END_FUNCTION_BLOCK

FUNCTION "FC_TPConveyorMapping" : Void
{ S7_Optimized_Access := 'TRUE' }
VERSION : 0.1
// ATTRIBUTES
// AUTO_NUMBER = True
// BLOCK_NUMBER = 30
// END_ATTRIBUTES
   VAR_INPUT
      iUDT_ConveyorStatus : "UDT_ConveyorStatus";
      iv_VfdStatus : Variant;
      iUDT_ConveyorInterface : "UDT_ConveyorInterface";
      iUDT_ConveyorConfiguration : "UDT_ConveyorConfiguration";
      is_ConveyorID : String;
   END_VAR

   VAR_OUTPUT
      qUDT_TPConveyorStatus : "UDT_ConveyorStatus";
      qUDT_TPConveyorInterface : "UDT_ConveyorInterface";
      qUDT_TPCommandState : "UDT_ConveyorCommand";   // Actual state of conveyor commands in DB_HMICommands
      qUDT_TPConveyorConfiguration : "UDT_ConveyorConfiguration";
      qs_TPSelectedConveyorName : String;
   END_VAR

   VAR_IN_OUT
      iqUDT_TPCommandButton : "UDT_TPManualControlButtons";
      iqUDT_ConveyorCommand : "UDT_ConveyorCommand";
      qUDT_TPVfdStatus : "UDT_VfdStatus";
   END_VAR

   VAR_TEMP
      tUDT_VfdStatus : "UDT_VfdStatus";
      tUDT_Ai2Status : "UDT_AixPlcFull4McoStatus";
      temp_ret_val : Int;
   END_VAR


BEGIN
	(*
	----------------------------------------------------------------------------------------

	Version history:
	Date        | Version   | Author        | Remark
	----------------------------------------------------------------------------------------
	18/10/2021  | 1.0       | S.Theocharis  | first release MHS TIA 16
	20/10/2021  | 1.1       | S.Theocharis  | change udt vfd status to variant
	03/06/2022  | 1.2       | M.Krystek     | change MOVE_BLK_VARIANT parameters
	21/02/2023  | 4.0       | F.Baten       | 4.0 Release TIA 17.5
	*)

	REGION 1 - Command Start

	    IF #iqUDT_TPCommandButton.ManualStart THEN
	        #iqUDT_ConveyorCommand.ManualStartStop := TRUE;
	        #iqUDT_TPCommandButton.ManualStart := False;
	    END_IF;

	END_REGION

	REGION 2 - Command Stop

	    IF #iqUDT_TPCommandButton.ManualStop THEN
	        #iqUDT_ConveyorCommand.ManualStartStop := FALSE;
	        #iqUDT_TPCommandButton.ManualStop := False;
	    END_IF;
	END_REGION

	REGION 3 - Command Nominal Speed

	    IF #iqUDT_TPCommandButton.ManualFullSpeed THEN
	        #iqUDT_ConveyorCommand.ManualFullSpeed := TRUE;
	        #iqUDT_TPCommandButton.ManualFullSpeed := False;
	    END_IF;
	END_REGION

	REGION 4 - Command Low Speed

	    IF #iqUDT_TPCommandButton.ManualLowSpeed THEN
	        #iqUDT_ConveyorCommand.ManualFullSpeed := FALSE;
	        #iqUDT_TPCommandButton.ManualLowSpeed := False;
	    END_IF;
	END_REGION

	REGION 5 - Command Reverse

	    IF #iqUDT_TPCommandButton.ManualReverse THEN
	        #iqUDT_ConveyorCommand.Reverse := NOT #iqUDT_ConveyorCommand.Reverse;
	        #iqUDT_ConveyorCommand.ManualStartStop := FALSE; //Stop always to avoid on the fly reverse
	        #iqUDT_TPCommandButton.ManualReverse := False;
	    END_IF;
	END_REGION

	REGION 6 - Command jog

	    #iqUDT_ConveyorCommand.ManualJog := #iqUDT_TPCommandButton.ManualJog;

	    IF #iqUDT_TPCommandButton.ManualJog THEN
	        #iqUDT_ConveyorCommand.ManualStartStop := FALSE;
	    END_IF;

	END_REGION

	REGION 7 - Status

	    #qUDT_TPCommandState := #iqUDT_ConveyorCommand;  //actual status of conveyor commands

	    #qUDT_TPConveyorStatus := #iUDT_ConveyorStatus; //conveyor status

	    //VFD status. Ignore Pulse roller
	    IF TypeOf(#iv_VfdStatus) = TypeOf(#tUDT_VfdStatus) THEN

	        #temp_ret_val := MOVE_BLK_VARIANT(SRC := #iv_VfdStatus,
	                                          COUNT := 1,
	                                          SRC_INDEX := 0,
	                                          DEST_INDEX := 0,
	                                          DEST => #qUDT_TPVfdStatus);

	    ELSE
	        #tUDT_VfdStatus.ErrorCode := #tUDT_VfdStatus.SubErrorCode := 0;
	        #qUDT_TPVfdStatus := #tUDT_VfdStatus;

	    END_IF;

	    //#q_TP_VFDStatus := #i_VFDStatus;

	    #qUDT_TPConveyorInterface := #iUDT_ConveyorInterface; //conveyor interface

	    #qs_TPSelectedConveyorName := #is_ConveyorID; //conveyor ID

	    #qUDT_TPConveyorConfiguration.Bi_Directional_Enable := #iUDT_ConveyorConfiguration.Bi_Directional_Enable; //read only bi directional enable bit from configuration


	END_REGION

END_FUNCTION

FUNCTION_BLOCK "FB_Induct"
TITLE = FB_Induct
{ S7_Optimized_Access := 'TRUE' }
AUTHOR : MHSE
FAMILY : Equipment
VERSION : 3.0
// ATTRIBUTES
// AUTO_NUMBER = True
// BLOCK_NUMBER = 14
// END_ATTRIBUTES
//Function block to control inducting the parcels to a merge conveyor
   VAR_INPUT
      iUDT_InductConfig { ExternalAccessible := 'False'; ExternalVisible := 'False'; ExternalWritable := 'False'} : "UDT_InductConfiguration";   //       Induct configuration parameters
      iUDT_MergeGenConfig { ExternalAccessible := 'False'; ExternalVisible := 'False'; ExternalWritable := 'False'} : "UDT_MergeGeneratorConfig";   //       Merge generator configuration parameters
      iUDT_MergeConvConfig { ExternalAccessible := 'False'; ExternalVisible := 'False'; ExternalWritable := 'False'} : "UDT_ConveyorCommonConfiguration";   //       Merge conveyor common configuration parameters
      iUDT_InductConvConfig { ExternalAccessible := 'False'; ExternalVisible := 'False'; ExternalWritable := 'False'} : "UDT_ConveyorConfiguration";   //       Induct conveyor configuration parameters
      iUDT_InductConvCommonStatus { ExternalAccessible := 'False'; ExternalVisible := 'False'; ExternalWritable := 'False'} : "UDT_CommonStatus";
      idi_PECEoSDistance { ExternalAccessible := 'False'; ExternalVisible := 'False'; ExternalWritable := 'False'} : DInt;   //       Distance between photo eye and the end of conveyor [mm]
      ii_Gin { ExternalAccessible := 'False'; ExternalVisible := 'False'; ExternalWritable := 'False'} : Int;   //       GIN from induct at photoeye position
      ix_SafetyOk { ExternalAccessible := 'False'; ExternalVisible := 'False'; ExternalWritable := 'False'} : Bool;   //       Safety is ok
      ix_inductEnable { ExternalAccessible := 'False'; ExternalVisible := 'False'; ExternalWritable := 'False'} : Bool := TRUE;   //      Enable the induct to make request
      ix_TrackingClear { ExternalAccessible := 'False'; ExternalVisible := 'False'; ExternalWritable := 'False'} : Bool;   //   Tracking area is clear of parcels
   END_VAR

   VAR_OUTPUT
      qx_ExternalRequestDieBack { ExternalAccessible := 'False'; ExternalVisible := 'False'; ExternalWritable := 'False'} : Bool;   // External request dieback
      qx_EnableAutoRecovey { ExternalAccessible := 'False'; ExternalVisible := 'False'; ExternalWritable := 'False'} : Bool;   // Request to enable auto recovery
   END_VAR

   VAR_IN_OUT
      iqs_TrackingData : Array[*] of Int;   //       Tracking data
      iqUDT_Merge : "UDT_Merge";   //       Gapgeneration data
      iqUDT_MergeInterface : "UDT_ConveyorInterface";
      iqUDT_InductInterface : "UDT_ConveyorInterface";
      iqUDT_HandShake : "UDT_ConveyorHandshake";
      iqa_ActualTimeData : Struct
         Offset : Int;
         Max_number_of_records : Int;
         Data {InstructionName := 'DTL'; LibVersion := '1.0'} : Array[0..99] of DTL;
      END_STRUCT;
   END_VAR

   VAR
      sR_TRIG_Displacement {InstructionName := 'R_TRIG'; LibVersion := '1.0'; ExternalAccessible := 'False'; ExternalVisible := 'False'; ExternalWritable := 'False'; S7_SetPoint := 'False'} : R_TRIG;   //       Signal rising edge displacement changed
      sR_TRIG_SetDelay {InstructionName := 'R_TRIG'; LibVersion := '1.0'; ExternalAccessible := 'False'; ExternalVisible := 'False'; ExternalWritable := 'False'; S7_SetPoint := 'False'} : R_TRIG;   //       Signal rising edge of parcel entering
      sR_TRIG_TIP {InstructionName := 'R_TRIG'; LibVersion := '1.0'; ExternalAccessible := 'False'; ExternalVisible := 'False'; ExternalWritable := 'False'; S7_SetPoint := 'False'} : R_TRIG;
      sR_TRIG_Enable {InstructionName := 'R_TRIG'; LibVersion := '1.0'; ExternalAccessible := 'False'; ExternalVisible := 'False'; ExternalWritable := 'False'; S7_SetPoint := 'False'} : R_TRIG;   //   Rising Edge of  Induct Enable signal
      sF_TRIG_sx_Parcel {InstructionName := 'F_TRIG'; LibVersion := '1.0'; ExternalAccessible := 'False'; ExternalVisible := 'False'; ExternalWritable := 'False'; S7_SetPoint := 'False'} : F_TRIG;   // Falling Trigger of sx_Parcel
      sdi_DelayReactivateReq { ExternalAccessible := 'False'; ExternalVisible := 'False'; ExternalWritable := 'False'} : DInt;   //       Actual counter delaying the reactivation request
      sdi_RunningEmpty { ExternalAccessible := 'False'; ExternalVisible := 'False'; ExternalWritable := 'False'} : DInt;   //       Actual counter distance running empty
      si_RequestLength { ExternalAccessible := 'False'; ExternalVisible := 'False'; ExternalWritable := 'False'} : Int;   //       Calculated length to be requested
      si_GINlength { ExternalAccessible := 'False'; ExternalVisible := 'False'; ExternalWritable := 'False'} : Int;   //       Length found in GIN DN or set beacuse of invalid length
      si_Gaplength { ExternalAccessible := 'False'; ExternalVisible := 'False'; ExternalWritable := 'False'} : Int;   //       Length for this parcel
      si_ArrayLengthFlexGap { ExternalAccessible := 'False'; ExternalVisible := 'False'; ExternalWritable := 'False'} : Int;   //       Size of the flexGapsize
      si_ArrayLengthTracking { ExternalAccessible := 'False'; ExternalVisible := 'False'; ExternalWritable := 'False'} : Int;   //       Size of the tracking array
      si_ArrayLengthFIFO { ExternalAccessible := 'False'; ExternalVisible := 'False'; ExternalWritable := 'False'} : Int;   //       Size of the FIFO
      si_DistanceToEnd { ExternalAccessible := 'False'; ExternalVisible := 'False'; ExternalWritable := 'False'} : Int;   //       Parcels distance to end of induct conveyor
      si_InductPoint { ExternalAccessible := 'False'; ExternalVisible := 'False'; ExternalWritable := 'False'} : Int;   //       Calculated induct point
      si_StartSearch { ExternalAccessible := 'False'; ExternalVisible := 'False'; ExternalWritable := 'False'} : Int;   //       Value declaring the start of the search area
      si_EndSearch { ExternalAccessible := 'False'; ExternalVisible := 'False'; ExternalWritable := 'False'} : Int;   //       Value declaring the end of the search area
      si_LoopCountFlexgap { ExternalAccessible := 'False'; ExternalVisible := 'False'; ExternalWritable := 'False'} : Int;   //       Loopcounter searching in configuration for a match for the parcellength
      si_LoopCountGapSearch { ExternalAccessible := 'False'; ExternalVisible := 'False'; ExternalWritable := 'False'} : Int;   //       Loopcounter searching in Trackingdata for a gap
      si_LoopCountCodeSearch { ExternalAccessible := 'False'; ExternalVisible := 'False'; ExternalWritable := 'False'} : Int;   //       Loopcounter searching for code -100
      si_LoopCountSyncSearch { ExternalAccessible := 'False'; ExternalVisible := 'False'; ExternalWritable := 'False'} : Int;   //       Loopcounter searching for code -100
      si_LoopCountFIFOSearch { ExternalAccessible := 'False'; ExternalVisible := 'False'; ExternalWritable := 'False'} : Int;   //       Loopcounter searching FIFO for request to remove
      si_LoopCountWriteGIN { ExternalAccessible := 'False'; ExternalVisible := 'False'; ExternalWritable := 'False'} : Int;   //       Loopcounter to write the GIN for the length of the parcel
      si_LastGIN { ExternalAccessible := 'False'; ExternalVisible := 'False'; ExternalWritable := 'False'} : Int;   //       Last processed GIN
      si_Flexgap { ExternalAccessible := 'False'; ExternalVisible := 'False'; ExternalWritable := 'False'} : Int;   //       Found flexible gapsize [cm]
      si_PosDataInSearchArea { ExternalAccessible := 'False'; ExternalVisible := 'False'; ExternalWritable := 'False'} : Int;   //       Length to wait to search for a gap
      si_WritePosition { ExternalAccessible := 'False'; ExternalVisible := 'False'; ExternalWritable := 'False'} : Int;   //       Position to write to in tracking
      si_Syncdifference { ExternalAccessible := 'False'; ExternalVisible := 'False'; ExternalWritable := 'False'} : Int;   //       Difference in positions pec and tracking
      si_SyncDistance { ExternalAccessible := 'False'; ExternalVisible := 'False'; ExternalWritable := 'False'} : Int;   //       Distance to perform the synchronisation in
      si_MergeRunLength { ExternalAccessible := 'False'; ExternalVisible := 'False'; ExternalWritable := 'False'} : Int;   //     Distance the merge conveyor has run when Inudct is waiting
      si_DelayDiebackLength { ExternalAccessible := 'False'; ExternalVisible := 'False'; ExternalWritable := 'False'} : Int;   //     length Run before applying die back [cm]
      si_TrackingPointer { ExternalAccessible := 'False'; ExternalVisible := 'False'; ExternalWritable := 'False'} : Int;   //   Tracking poitner to search in the tracking
      sx_Sync { ExternalAccessible := 'False'; ExternalVisible := 'False'; ExternalWritable := 'False'} : Bool;   //       Code search to synchronise
      sx_ConfigError { ExternalAccessible := 'False'; ExternalVisible := 'False'; ExternalWritable := 'False'} : Bool;   //       Error in the configuration
      sx_FindLength { ExternalAccessible := 'False'; ExternalVisible := 'False'; ExternalWritable := 'False'} : Bool;   //       Find the length of the new parcel
      sx_Parcel { ExternalAccessible := 'False'; ExternalVisible := 'False'; ExternalWritable := 'False'} : Bool;   //       The parcel is present an not yet handled completely
      sx_GapRequested { ExternalAccessible := 'False'; ExternalVisible := 'False'; ExternalWritable := 'False'} : Bool;   //       The request is done for the latest parcel
      sx_SearchGapInTracking { ExternalAccessible := 'False'; ExternalVisible := 'False'; ExternalWritable := 'False'} : Bool;   //       True = Search for space in tracking to induct without merge generation
      sx_LastCodeNeg { ExternalAccessible := 'False'; ExternalVisible := 'False'; ExternalWritable := 'False'} : Bool;   //       True = Last found code was a negative one
      sx_FreeGapAvailable { ExternalAccessible := 'False'; ExternalVisible := 'False'; ExternalWritable := 'False'} : Bool;   //       There is a free space found, big enough to insert the parcel
      sx_ValidWindowCodeFound { ExternalAccessible := 'False'; ExternalVisible := 'False'; ExternalWritable := 'False'} : Bool;   //       There is a valid window code found
      sx_CodeAtposition { ExternalAccessible := 'False'; ExternalVisible := 'False'; ExternalWritable := 'False'} : Bool;
      sx_InductEnable { ExternalAccessible := 'False'; ExternalVisible := 'False'; ExternalWritable := 'False'} : Bool;   //       The parcel is enabled to induct
      sx_DiebackInductConveyor { ExternalAccessible := 'False'; ExternalVisible := 'False'; ExternalWritable := 'False'} : Bool;   //       Memory to stop the induct conveyor
      sx_Hold { ExternalAccessible := 'False'; ExternalVisible := 'False'; ExternalWritable := 'False'} : Bool;   //       Hold inducting
      sx_Active { ExternalAccessible := 'False'; ExternalVisible := 'False'; ExternalWritable := 'False'} : Bool;
      sx_EnableAutoRecovery { ExternalAccessible := 'False'; ExternalVisible := 'False'; ExternalWritable := 'False'} : Bool;   //     Enable Auto Recovery for Induct
      sx_RecoveryRequest { ExternalAccessible := 'False'; ExternalVisible := 'False'; ExternalWritable := 'False'} : Bool;
   END_VAR

   VAR CONSTANT
      ci_SearchArea : Int := 3;
   END_VAR


BEGIN
	(*
	----------------------------------------------------------------------------------------

	Version history:
	Date        | Version   | Author        | Remark
	----------------------------------------------------------------------------------------
	24/09/2019  | 1.0       | F.Baten       | first release TIA 15.1
	31/10/2019  | 1.1       | F.Baten       | qi_SpeedSetpoint changed to int because of conveyor interface change
	12/11/2019  | 3.0       | P.Majka       | 3.0 MHS library release TIA 15.1
	07/01/2020  | 3.1       | F.Baten       | Changed RequestInFifo to be handshaking
	                                        | Merged region 4.3 and 4.4
	09/01/2020  | 3.2       | F.Baten       | Removed speed calculation
	14/01/2020  | 3.3       | F.Baten       | Removed global FIFO full signal as it was not generated and made it local
	14/01/2020  | 3.4       | F.Baten       | Changed displacement detection equal to 0 and not to be 1 as it can also be bigger
	            | 3.5       |               | Renamed ii_PEC_EoSDistance to idi_PEC_EoSDistance
	15/01/2020  | 3.6       | L.Klar        | GIN record structure updated, parcel length remapped
	23/01/2020  | 3.7       | F.Baten       | Added reset when parcel is at end of conveyor but for some reason not detected
	                                          Modified dieback: alsways goto dieback when parcel is handled
	18/02/2020  | 3.8       | F.Baten       | Modified "Search 1: Gap '0'" , added +1 to wait to search again.
	15/10/2020  | 3.9       | F.Baten       | Reqactivation request: added if active to keep active
	                                          removed displacement check out of search
	20/05/2021  | 3.10      | M.Singh       | Enabled Auto Recovery based on the displacemt on Merge
	20/04/2022  | 3.11      | M.Piela       | Added Auto recovery output
	24/05/2022  | 3.12      | M.Roijen      | Changed FOR loop region 5.2 copy gin to tracking (add -1).
	22/07/2022  | 3.13      | M.Piela       | Reset the sx_Active and set dieback induct on falling edge of sx_Parcel instead of rising edge of TIP.
	21/02/2023  | 4.0       | F.Baten       | 4.0 Release TIA 17.5
	*)

	REGION 1 - New GIN received
	    // When the new GIN is received:
	    // - first save the GIN and set/reset statuses
	    // - calculate the requested length for this parcel
	    // - requeset a gap for this parcel

	    REGION 1.1 - New gin received is NOT equal TO '0' AND NOT equal TO last gin
	        //#s_R_TRIG_TIP(CLK := #iq_UDT_HandShake.TIP);
	        // IF #ii_Gin <> 0 AND #ii_Gin <> #si_LastGIN AND NOT #iq_UDT_HandShake.TIP AND NOT #s_F_TRIG_TIP.Q

	        IF #ii_Gin <> 0 AND #ii_Gin <> #si_LastGIN AND #ix_inductEnable
	        THEN
	            #sx_FindLength := FALSE;                                                    // To set length for a flexible gap
	            #sx_GapRequested := FALSE;                                                  // To initiate length calculation for gap and request the gap to FIFO
	            #sx_DiebackInductConveyor := TRUE;                                             // Activate dieback to stop the conveyor while waiting on a gap
	            #sx_Sync := FALSE;                                                          // Sync speed is not calculated
	            #sx_Parcel := TRUE;                                                         // Activate the induct search
	            #sx_Active := TRUE;                                                         // The parcel is not transferred to the next conveyor
	            #si_LastGIN := #ii_Gin;                                                     // Memorise
	            #si_DistanceToEnd := DINT_TO_INT(#idi_PECEoSDistance) / 10;                // Actual distance to end (in tracking array units)
	            #si_GINlength := DINT_TO_INT("DB_GIN".GIN[#si_LastGIN].General.Length);     // set length
	            IF #si_GINlength = 0
	            THEN
	                #si_GINlength := #iUDT_InductConfig.MaxParcelSize / 10;
	            END_IF;

	            IF #sx_RecoveryRequest
	            THEN

	                #si_DistanceToEnd := #iUDT_InductConfig.ParcelStopPositionAutoRecovery;                                                     // Actual distance to end (in tracking array units)
	                #si_GINlength := (#iUDT_InductConfig.MaxParcelSize / 10) + #iUDT_InductConfig.RecoveryAdditionalGap;
	                #sx_RecoveryRequest := FALSE;
	            END_IF;

	        END_IF;

	        // There is a parcel on the inductconveyor but it had no GIN (not even UFO)
	        IF (#iqUDT_HandShake.RTS                                                       // If Induct is ready to Send
	            OR #iUDT_InductConvCommonStatus.Dieback)                                   // Or is in die back
	            AND NOT #sx_Active                                                          // And Induct is not active
	            AND #ix_inductEnable
	        THEN
	            #si_MergeRunLength := #si_MergeRunLength - #iqUDT_MergeInterface.Displacement;
	        ELSE
	            #si_MergeRunLength := #iUDT_InductConfig.DistanceRunBeforeAutoRecovery;
	        END_IF;

	        #sx_EnableAutoRecovery := FALSE;

	        IF #si_MergeRunLength <= 0
	        THEN
	            #sx_EnableAutoRecovery := True;
	            #si_MergeRunLength := #iUDT_InductConfig.DistanceRunBeforeAutoRecovery;
	        END_IF;

	        #sR_TRIG_Enable(CLK := #ix_inductEnable);

	        IF #sx_EnableAutoRecovery                                                     // Make a new request to autorecover
	            OR (#sR_TRIG_Enable.Q
	            AND NOT #ix_TrackingClear)
	        THEN
	            #sx_FindLength := FALSE;                                                    // To set length for a flexible gap
	            #sx_GapRequested := FALSE;                                                  // To initiate length calculation for gap and request the gap to FIFO
	            #sx_DiebackInductConveyor := TRUE;                                             // Activate dieback to stop the conveyor while waiting on a gap
	            #sx_Sync := FALSE;                                                          // Sync speed is not calculated
	            #sx_Parcel := TRUE;                                                         // Activate the induct search
	            #sx_Active := TRUE;                                                         // The parcel is not transferred to the next conveyor
	            #si_LastGIN := -50;                                                         // Memorise
	            #si_DistanceToEnd := #iUDT_InductConfig.ParcelStopPositionAutoRecovery;                                                     // Actual distance to end (in tracking array units)
	            #si_GINlength := (#iUDT_InductConfig.MaxParcelSize / 10) + #iUDT_InductConfig.RecoveryAdditionalGap;
	            #sx_RecoveryRequest := TRUE;



	            // temp code
	            #iqa_ActualTimeData.Data[#iqa_ActualTimeData.Offset] := "DB_Time".ActualTimeDTL;
	            #iqa_ActualTimeData.Offset := #iqa_ActualTimeData.Offset + 1;
	        END_IF;

	        #qx_EnableAutoRecovey := #sx_EnableAutoRecovery;

	        IF #iqa_ActualTimeData.Offset = #iqa_ActualTimeData.Max_number_of_records
	        THEN
	            #iqa_ActualTimeData.Offset := 1;
	        END_IF;


	    END_REGION

	    REGION 1.2 - Calculate the required gap depending on the mode
	        CASE #iUDT_InductConfig.GapMode OF

	            1:  // Gap is Head to head
	                #si_RequestLength := #iUDT_InductConfig.GapHeadToHead;
	                #si_Gaplength := #si_RequestLength - #si_GINlength;
	                #sx_FindLength := TRUE;                                                 // New GIN length is set

	            2:  // Gap is parcel length + tail to head (fixed)
	                #si_RequestLength := #si_GINlength + #iUDT_InductConfig.GapTailToHead;
	                #si_Gaplength := #iUDT_InductConfig.GapTailToHead;
	                #sx_FindLength := TRUE;                                                 // New GIN length is set

	            3:  // Gap is parcel length + gap depending on length of parcel
	                IF NOT #sx_FindLength
	                THEN
	                    #si_ArrayLengthFlexGap := "FC_GetNrOfArrayEl"(#iUDT_InductConfig.FlexGap); // Determine size of search area
	                    FOR #si_LoopCountFlexgap := 1 TO #si_ArrayLengthFlexGap BY 1 DO                   // Set the loopcounter
	                        #si_Flexgap := #iUDT_InductConfig.MinParcelSize / 10;      // set minimal gapsize
	                        IF #si_GINlength < #iUDT_InductConfig.FlexGap[#si_LoopCountFlexgap]."Maximal length"
	                        THEN
	                            #si_Flexgap := #iUDT_InductConfig.FlexGap[#si_LoopCountFlexgap].Gap;
	                            EXIT;
	                        END_IF;
	                    END_FOR;
	                    #sx_FindLength := TRUE;                                             // New GIN length is calculated
	                END_IF;
	                #si_RequestLength := #si_GINlength + #si_Flexgap;
	                #si_Gaplength := #si_Flexgap;
	                ;

	        END_CASE;
	    END_REGION

	    REGION 1.3 - General
	        // When the transfer is finished set the induct to dieback

	        // IF #s_R_TRIG_TIP.Q  AND NOT #sx_Parcel
	        IF #sF_TRIG_sx_Parcel.Q
	        THEN
	            //     #si_DelayDiebackLength := #i_UDT_InductConfig.MinParcelSize;

	            // END_IF;

	            // IF #si_DelayDiebackLength > 0
	            // THEN
	            //     #si_DelayDiebackLength := #si_DelayDiebackLength - #iq_UDT_InductInterface.Displacement;
	            // END_IF;
	            // IF #si_DelayDiebackLength <= 0
	            // THEN
	            #sx_DiebackInductConveyor := TRUE;                                             // Activate dieback to stop the conveyor while waiting on a gap
	            #sx_Active := FALSE;                                                            // The parcel is now transferred to the next conveyor
	        END_IF;
	        //  #s_R_TRIG_TIP(CLK := #iq_UDT_HandShake.TIP);
	        #sF_TRIG_sx_Parcel(CLK := #sx_Parcel);
	        // When safety is not ok, load the run empty distance
	        IF NOT #ix_SafetyOk
	        THEN
	            #sdi_RunningEmpty := #iUDT_InductConfig.RunEmptyDistance;
	        END_IF;

	        // Hold inducting functions while mergeconveyor runs empty
	        #sx_Hold := (#sdi_RunningEmpty <> 0);

	        // Check every change of the merge conveyor's displacement
	        #sR_TRIG_Displacement(CLK := #iqUDT_MergeInterface.Displacement = 0);             // The merge conveyor has had displacement
	    END_REGION
	END_REGION

	REGION 2 - Request
	    REGION 2.1 - FIFO request
	        // request gap/window for induct
	        IF #sx_Parcel
	            AND NOT #sx_Hold                                                            // Holding all actions
	            AND NOT #sx_GapRequested                                                    // Gap is NOT requested
	            AND NOT #iqUDT_Merge.RequestInFIFO[#iUDT_InductConfig.Induct_Number]      // Requeset is in FIFO
	            AND NOT #iqUDT_Merge.GenerationInactive                                    // Generation is active
	            AND NOT #iUDT_InductConfig.SearchOnly                                      // Only searching for a gap
	            AND NOT (#iqUDT_Merge.LastUsed = #iqUDT_Merge.MaxNumberofEntries)         // The FIFO is full
	        THEN
	            #iqUDT_Merge.LastUsed += 1;                                                // Increase
	            #iqUDT_Merge.RequestInFIFO[#iUDT_InductConfig.Induct_Number] := TRUE;     // Memorise
	            #iqUDT_Merge.FIFO[#iqUDT_Merge.LastUsed].InductNumber := #iUDT_InductConfig.Induct_Number;   // Write the induct number
	            #iqUDT_Merge.FIFO[#iqUDT_Merge.LastUsed].GapSize := DINT_TO_INT(#si_RequestLength);           // Write the requested length
	            #iqUDT_Merge.FIFO[#iqUDT_Merge.LastUsed].RemoveEntry := FALSE;                                // Reset remove bit
	            #sx_GapRequested := TRUE;                                                   // Gap is requested
	        END_IF;
	    END_REGION

	    REGION 2.2 - Reactivation of merge generator block
	        // If not in searchmode, every time a parcel enters, the waiting distance is set
	        IF NOT #iUDT_InductConfig.SearchOnly
	        THEN
	            #sR_TRIG_SetDelay(CLK := #sx_Parcel);
	        ELSE
	            #sR_TRIG_SetDelay.Q := FALSE;
	        END_IF;

	        IF #sR_TRIG_SetDelay.Q
	        THEN
	            #sdi_DelayReactivateReq := #iUDT_InductConfig.ReactivationRequestDelay / 10;
	        END_IF;

	        // Reactivation request merge generator block
	        // In gapmode 3 the generator is not allowed to deactivate
	        #iqUDT_Merge.ReactivateReq :=
	        ((#sdi_DelayReactivateReq = 0)
	        AND #sx_Parcel
	        AND #iqUDT_Merge.GenerationInactive
	        AND NOT #iUDT_InductConfig.SearchOnly)
	        OR (#iUDT_InductConfig.GapMode = 3)
	        OR #iqUDT_Merge.ReactivateReq;

	    END_REGION
	END_REGION

	REGION 3 - Displacement

	    REGION 3.1 - Track induct point
	        IF #iqUDT_Merge.TrackingPointerForInduct[#iUDT_InductConfig.Induct_Number] > 0
	        THEN
	            #iqUDT_Merge.TrackingPointerForInduct[#iUDT_InductConfig.Induct_Number] -= #iqUDT_MergeInterface.Displacement;
	            IF #iqUDT_Merge.TrackingPointerForInduct[#iUDT_InductConfig.Induct_Number] < 0                                              // check if the value does not go negative
	            THEN
	                #iqUDT_Merge.TrackingPointerForInduct[#iUDT_InductConfig.Induct_Number] := 0;
	            END_IF;
	        END_IF;
	    END_REGION

	    REGION 3.2 - Wait distance
	        // If a value is found during the search for an empty position, the position of the tracking is saved.
	        // This value is decreased by displacement to wait for the next time the tracking should be searched again.
	        IF #si_PosDataInSearchArea > 0
	        THEN
	            #si_PosDataInSearchArea -= #iqUDT_MergeInterface.Displacement;
	            IF #si_PosDataInSearchArea < 0                                              // check if the value does not go negative
	            THEN
	                #si_PosDataInSearchArea := 0;
	            END_IF;
	        END_IF;

	        // The parcel is waiting to be inducted
	        IF #sdi_DelayReactivateReq > 0 AND NOT #sx_Hold
	        THEN
	            #sdi_DelayReactivateReq -= #iqUDT_MergeInterface.Displacement;
	            IF #sdi_DelayReactivateReq < 0                                              // check if the value does not go negative
	            THEN
	                #sdi_DelayReactivateReq := 0;
	            END_IF;
	        END_IF;

	        // the distance to the end of the induct conveyor, the parcel travelling on the induct conveyor
	        IF #si_DistanceToEnd > 0 // AND #iq_UDT_InductInterface.RunFwd
	        THEN
	            #si_DistanceToEnd -= #iqUDT_InductInterface.Displacement;
	            IF #si_DistanceToEnd < 0                                                    // check if the value does not go negative
	            THEN
	                #si_DistanceToEnd := 0;
	            END_IF;
	        END_IF;

	        // the distance to run empty
	        IF #sdi_RunningEmpty > 0
	        THEN
	            #sdi_RunningEmpty -= #iqUDT_MergeInterface.Displacement;
	            IF #sdi_RunningEmpty < 0                                                    // check if the value does not go negative
	            THEN
	                #sdi_RunningEmpty := 0;
	            END_IF;
	        END_IF;
	    END_REGION
	END_REGION

	REGION 4 - Search position
	    REGION 4.1 - General
	        // When the generator is not active and there is no active request
	        // search for gap which is completely empty only when generator is switched off or the mode is search only
	        #sx_SearchGapInTracking := #iqUDT_Merge.GenerationInactive
	        OR #iUDT_InductConfig.SearchOnly;

	        // set the Induct position to cm and a moving box while searching is a moving inductpoint
	        #si_InductPoint := (#iUDT_InductConfig.Induct_Position / 10);//- ((DINT_TO_INT(#idi_PEC_EoSDistance) / 10) - #si_DistanceToEnd);
	        // #si_InductPoint := (#i_UDT_InductConfig.Induct_Position / 10) - ((DINT_TO_INT(#idi_PEC_EoSDistance) / 10));
	        // In mode 3 the gap in front of the parcel is determined by the size of the parcel, this means the gap is leading. This is needed for some devices such as weighing scales.
	        // To get the gap in front of the parcel, the point of detecting the requested code is delayed by the gapsize.
	        // When the parcel starts now, it should be the length of the gap after the detected code. When writing in tracking the GIN is written aligned with the parcel, in the back of the window.
	        // So, it moves the inductionpoint forwards in the tracking (downstream) with the parcels Flexgap.

	        CASE #iUDT_InductConfig.GapMode OF
	            3:
	                #si_InductPoint -= #si_Flexgap;
	        END_CASE;

	    END_REGION

	    REGION 4.2 - Search 1: Gap '0'
	        // 1: Search for a gap (tracking is filled with '0')
	        // When a value is found in the tracking, we do not have to search again until that value has passed.
	        //
	        // search from  :  Induct position forward (gaptailtohead) because the last parcel can just have passed the position
	        // to           :  induct position + length of the parcel and its gap tail to next head
	        //
	        IF #sx_Parcel                                                                   // A parcel is present
	            //    AND #s_R_TRIG_Displacement.Q                                                // There was a displacement
	            AND #si_PosDataInSearchArea = 0                                             // No wait length
	            AND #sx_SearchGapInTracking                                                 // Search for empty gap is activated
	            AND NOT #sx_Hold                                                            // merge conveyor is available
	        THEN
	            #si_StartSearch := (#si_InductPoint - #iUDT_InductConfig.GapTailToHead);
	            #si_EndSearch := (#si_InductPoint + DINT_TO_INT(#si_RequestLength));
	            FOR #si_LoopCountGapSearch := #si_StartSearch TO #si_EndSearch BY 1 DO

	                IF (#iqs_TrackingData[#si_LoopCountGapSearch] <> 0)                       // There is a value in the tracking area
	                THEN
	                    IF #iqs_TrackingData[#si_LoopCountGapSearch] < 0                      // the value was a negative value so wait for that to pass
	                    THEN
	                        #si_PosDataInSearchArea := #si_LoopCountGapSearch - #si_StartSearch + 1; // Save the distance added by 1 to wait to search again on the next position
	                        EXIT;
	                    END_IF;

	                    IF #iqs_TrackingData[#si_LoopCountGapSearch] > 0                      // The value is positive: GIN
	                    THEN
	                        #si_PosDataInSearchArea := #si_LoopCountGapSearch - #si_StartSearch + 1;  // As long as the GIN is found the wait distance is increased
	                    END_IF;
	                END_IF;
	            END_FOR;

	            IF #si_PosDataInSearchArea = 0                                          // memory is empty after search
	            THEN
	                #sx_FreeGapAvailable := True;                                       // There is a gap, large enough to put the parcel in
	                #si_WritePosition := #si_InductPoint;
	            END_IF;
	        END_IF;
	    END_REGION



	    REGION 4.3 - Search 2: code -100, -10(x) or -200-
	        IF #sx_Parcel                                                               // A parcel is present
	            //       AND #s_R_TRIG_Displacement.Q                                            // There was a displacement
	            AND NOT #sx_SearchGapInTracking                                         // Search for empty gap is not activated
	            AND NOT #sx_Hold                                                        // merge conveyor is available
	        THEN
	            // 2: search for the code -100 around the induct position within search area, displacement can be more than 1
	            //    search for the code -200- , code (-)200 + size of the gap . This was a gap requested but not used, the value over 200 indicates the size

	            #sx_ValidWindowCodeFound := FALSE;                                      // reset the memory
	            FOR #si_LoopCountCodeSearch := #si_InductPoint TO (#si_InductPoint + #ci_SearchArea) BY 1 DO

	                IF (#iqs_TrackingData[#si_LoopCountCodeSearch] = -100)                    // If the value is -100
	                    OR (#iqs_TrackingData[#si_LoopCountCodeSearch] = (-100 - (#iUDT_InductConfig.Induct_Number)))
	                THEN
	                    #sx_ValidWindowCodeFound := TRUE;                               // Set the memory
	                    #si_WritePosition := #si_LoopCountCodeSearch;                         // save the position to write to
	                    EXIT;                                                           // Stop searchloop

	                ELSIF (#iqs_TrackingData[#si_LoopCountCodeSearch] <= -200)               // If the value is less than -200 (a not used gap)
	                    AND ((#iqs_TrackingData[#si_LoopCountCodeSearch] + 200) * -1) > #si_RequestLength // The length of this gap is bigger than the one which is needed
	                THEN
	                    #sx_ValidWindowCodeFound := TRUE;                               // Set the memory
	                    #si_WritePosition := #si_LoopCountCodeSearch;                         // save the position to write to
	                    EXIT;                                                           // Stop searchloop
	                END_IF;
	            END_FOR;
	        END_IF;
	    END_REGION

	END_REGION

	REGION 5 - Do induct

	    // enable induct
	    #sx_InductEnable :=
	    #sx_FreeGapAvailable                                                            // There is a gap, large enough to put the parcel in
	    OR #sx_ValidWindowCodeFound;                                                    // A valid induct code is found

	    IF #sx_Parcel AND #sx_InductEnable
	    THEN

	        // check if position can be written in tracking array
	        #si_ArrayLengthTracking := "FC_GetNrOfArrayEl"(#iqs_TrackingData);          // Determine size of search area
	        #sx_ConfigError := (#si_WritePosition + #si_RequestLength) > #si_ArrayLengthTracking;
	        #si_DistanceToEnd := 0;                                                     // Release conveyors nominal speed

	        REGION 5.1 - Update FIFO
	            // If the RequestIsInFIFO is still true, it  means the merge generator did not handle this request yet.
	            // Now the FIFO is searched for the induct number.
	            // On this entry the bit remove is set and also the Remove hanshake is set to indicate to the merge generator an entry has to be removed

	            IF #iqUDT_Merge.RequestInFIFO[#iUDT_InductConfig.Induct_Number]
	            THEN
	                #si_ArrayLengthFIFO := "FC_GetNrOfArrayEl"(#iqUDT_Merge.FIFO);     // Determine size of search area
	                FOR #si_LoopCountFIFOSearch := 0 TO (#si_ArrayLengthFIFO - 1) BY 1 DO
	                    IF #iqUDT_Merge.FIFO[#si_LoopCountFIFOSearch].InductNumber = #iUDT_InductConfig.Induct_Number
	                    THEN
	                        #iqUDT_Merge.FIFO[#si_LoopCountFIFOSearch].RemoveEntry := TRUE;
	                        #iqUDT_Merge.Remove := TRUE;
	                        EXIT;
	                    END_IF;
	                END_FOR;
	                #iqUDT_Merge.RequestInFIFO[#iUDT_InductConfig.Induct_Number] := False;
	            END_IF;
	        END_REGION

	        REGION 5.2 - Copy GIN to tracking
	            // write GIN to merge conveyor tracking for the length of the parcel
	            FOR #si_LoopCountWriteGIN := #si_WritePosition TO (#si_WritePosition + #si_RequestLength - 1) BY 1 DO
	                #iqs_TrackingData[#si_LoopCountWriteGIN] := 0;
	            END_FOR;
	            CASE #iUDT_InductConfig.GapMode OF
	                1, 2: // write data leading
	                    FOR #si_LoopCountWriteGIN := #si_WritePosition TO (#si_WritePosition + #si_GINlength) BY 1 DO
	                        #iqs_TrackingData[#si_LoopCountWriteGIN] := #si_LastGIN;
	                    END_FOR;
	                3: // write gap leading
	                    FOR #si_LoopCountWriteGIN := #si_WritePosition + #si_Gaplength TO (#si_WritePosition + #si_RequestLength) BY 1 DO
	                        #iqs_TrackingData[#si_LoopCountWriteGIN] := #si_LastGIN;
	                    END_FOR;
	            END_CASE;
	        END_REGION

	        REGION 5.3 - Update request in tracking
	            // reset the request in the tracking if the request is there
	            IF #iqs_TrackingData[#iqUDT_Merge.TrackingPointerForInduct[#iUDT_InductConfig.Induct_Number]] = (-100 - (#iUDT_InductConfig.Induct_Number))
	            THEN
	                CASE #iUDT_InductConfig.GapMode OF
	                    1:  // All gaps are head to headsize: reserved window code to be overwritted with fixed window code -100
	                        #iqs_TrackingData[#iqUDT_Merge.TrackingPointerForInduct[#iUDT_InductConfig.Induct_Number]] := -100;
	                    2, 3:  // Mark as NOT used (-200) AND give the gapsize as was requested
	                        #iqs_TrackingData[#iqUDT_Merge.TrackingPointerForInduct[#iUDT_InductConfig.Induct_Number]] := (-200 - #si_RequestLength);
	                END_CASE;
	            END_IF;
	        END_REGION

	        REGION 5.4 - Reset data (end of cycle)
	            // reset the inducting data
	            #iqUDT_Merge.TrackingPointerForInduct[#iUDT_InductConfig.Induct_Number] := 0;     // reset the pointer, the parcel is handled
	            #sx_FreeGapAvailable := FALSE;                                              // There is a gap, large enough to put the parcel in
	            #sx_ValidWindowCodeFound := FALSE;                                          // A free induct code is found
	            #sx_DiebackInductConveyor := FALSE;                                            // Release the parcel
	            #sx_GapRequested := FALSE;                                                  // To initiate length calculation for gap and request the gap to FIFO
	            #sx_Parcel := FALSE;                                                        // The parcel is handled
	        END_REGION
	    END_IF;

	    REGION 5.5 - Missed request, do again
	        IF #sx_GapRequested = TRUE                                                      // Gap is requested
	            AND NOT #iqUDT_Merge.RequestInFIFO[#iUDT_InductConfig.Induct_Number]      // No request in FIFO
	            AND #iqUDT_Merge.TrackingPointerForInduct[#iUDT_InductConfig.Induct_Number] = 0   // pointer elapsed
	        THEN
	            #sx_GapRequested := FALSE;                                                  // Reset the gap was requested and do request again
	        END_IF;
	    END_REGION
	END_REGION

	REGION 6 - Conveyor

	    // Stop the induct conveyor
	    #qx_ExternalRequestDieBack := #sx_DiebackInductConveyor;
	END_REGION

	//#iq_UDT_Merge.ReactivateReq := true;
END_FUNCTION_BLOCK

FUNCTION_BLOCK "FB_AirPressureFault"
{ S7_Optimized_Access := 'TRUE' }
VERSION : 0.1
// ATTRIBUTES
// AUTO_NUMBER = True
// BLOCK_NUMBER = 3
// END_ATTRIBUTES
   VAR_INPUT
      ix_AirPressureSwitch { ExternalAccessible := 'False'; ExternalVisible := 'False'; ExternalWritable := 'False'} : Bool;   // Air Pressure switch input
   END_VAR

   VAR_OUTPUT
      qUDT_HMIStatus : "UDT_AirPressureSwitchStatus";   // Air pressure switch  fault status
   END_VAR

   VAR_IN_OUT
      iqUDT_EquipmentControl : "UDT_EquipmentControl";   // Equipment control structure
   END_VAR

   VAR
      sx_AirPressureFault { ExternalAccessible := 'False'; ExternalVisible := 'False'; ExternalWritable := 'False'} : Bool;   // When TRUE air pressure fault is active
   END_VAR


BEGIN
	(*
	----------------------------------------------------------------------------------------

	Version history:
	Date        | Version   | Author        | Remark
	----------------------------------------------------------------------------------------
	19/07/2022  | 0.1       | M.Piela       | first release MHS TIA 16.0
	21/02/2023  | 4.0       | F.Baten       | 4.0 Release TIA 17.5
	*)

	REGION 1 - Reset encoder error

	    IF #iqUDT_EquipmentControl.Command.Reset THEN
	        #sx_AirPressureFault := FALSE;
	    END_IF;

	END_REGION

	REGION 2 - Set air pressure switch error

	    IF NOT #ix_AirPressureSwitch
	    THEN
	        #sx_AirPressureFault := TRUE;
	    END_IF;

	END_REGION

	REGION 3 - Status

	    #qUDT_HMIStatus.Specific.AirPressureOK := NOT #sx_AirPressureFault;

	    IF #sx_AirPressureFault
	    THEN
	        #qUDT_HMIStatus.Status := "DB_HMIStatusConfiguration".Error;
	    END_IF;

	    IF NOT #sx_AirPressureFault
	    THEN
	        #qUDT_HMIStatus.Status := "DB_HMIStatusConfiguration".AutoON;
	    END_IF;

	END_REGION

END_FUNCTION_BLOCK

FUNCTION_BLOCK "FB_OnOffDevices"
TITLE = FB_OnOffDevices
{ S7_Optimized_Access := 'TRUE' }
AUTHOR : MHSE
FAMILY : GeneralSystemFunctions
VERSION : 3.0
// ATTRIBUTES
// AUTO_NUMBER = True
// BLOCK_NUMBER = 19
// END_ATTRIBUTES
//Function block to enable and disable profinet devices.
   VAR_INPUT
      ix_Simulation { ExternalAccessible := 'False'; ExternalVisible := 'False'; ExternalWritable := 'False'} : Bool;   // Simulation on or off
   END_VAR

   VAR_OUTPUT
      qx_Done { ExternalAccessible := 'False'; ExternalVisible := 'False'; ExternalWritable := 'False'} : Bool;   // Operation done
      qx_Error { ExternalAccessible := 'False'; ExternalVisible := 'False'; ExternalWritable := 'False'} : Bool;   // Collective error output
   END_VAR

   VAR_IN_OUT
      iqa_ProfinetNetworks : Array[*] of "UDT_ProfinetNetwork";   // Profinet networks structure
   END_VAR

   VAR
      sR_TRIG_StartSim {InstructionName := 'R_TRIG'; LibVersion := '1.0'; ExternalAccessible := 'False'; ExternalVisible := 'False'; ExternalWritable := 'False'; S7_SetPoint := 'False'} : R_TRIG;   // Rising edge simulation bit
      sF_TRIG_StartSim {InstructionName := 'F_TRIG'; LibVersion := '1.0'; ExternalAccessible := 'False'; ExternalVisible := 'False'; ExternalWritable := 'False'; S7_SetPoint := 'False'} : F_TRIG;   // Falling edge simulation bit
      si_ActualStatus { ExternalAccessible := 'False'; ExternalVisible := 'False'; ExternalWritable := 'False'} : Int;   // Status structure
      si_Mode { ExternalAccessible := 'False'; ExternalVisible := 'False'; ExternalWritable := 'False'} : USInt;   // Simulation mode 1 - simulation off 2 - simulation on
      sx_OperationReq { ExternalAccessible := 'False'; ExternalVisible := 'False'; ExternalWritable := 'False'} : Bool;   // Operation required
   END_VAR

   VAR_TEMP
      ti_LoopCounterDevices : Int;   // Temporary counter of "for" loop
      ti_LoopCounterNetworks : Int;   // Temporary counter of "for" loop
      ti_NrOfProfinetDevices : Int;   // Number of profinet devices
      ti_NrOfNetworks : Int;   // Number of Profinet networks
      tx_Busy : Bool;   // D_ACT_DP busy
   END_VAR


BEGIN
	(*
	----------------------------------------------------------------------------------------

	Version history:
	Date        | Version   | Author        | Remark
	----------------------------------------------------------------------------------------
	24/05/2019  | 0.1       | K.Pokorski    | first release MHS TIA 15.1
	24/06/2019  | 0.2       | L.Klar        | Status running added
	19/07/2019  | 0.5       | L.Klar        | Status handling changed, output qx_Done added
	24/07/2019  | 2.0       | L.Klar        | 2.0 MHS library release TIA 15.1
	14/08/2019  | 2.1       | K.Pokorski    | Devices HW_ID extract deleted
	26/08/2019  | 2.2       | K.Pokorski    | Comments adjusted
	30/09/2019  | 2.3       | K.Pokorski    | Network seach started from 1 instead 0
	04/11/2019  | 2.4       | L.Klar        | First scan bit changed from memory bit to DB variable
	12/11/2019  | 3.0       | P.Majka       | 3.0 MHS library release TIA 15.1
	21/02/2023  | 4.0       | F.Baten       | 4.0 Release TIA 17.5
	*)

	REGION 1 – Mode selection

	    #sR_TRIG_StartSim(CLK := #ix_Simulation);

	    #sF_TRIG_StartSim(CLK := #ix_Simulation);

	    // Set operation request and operation mode (2 - devices deactivation) (1 - devices activation) when the simulation input has changed or the first PLC scan occurred
	    IF (#sR_TRIG_StartSim.Q            // Device activation required
	        OR #sF_TRIG_StartSim.Q         // Device deactivation required
	        OR "DB_Memory".FirstScan)       // First PLC scan occured
	    THEN

	        #sx_OperationReq := TRUE;

	        IF (NOT #ix_Simulation)                                             // Simulation turned off
	        THEN

	            #si_Mode := 1;

	        END_IF;

	        IF (#ix_Simulation)                                                 // Simulation turned on
	        THEN

	            #si_Mode := 2;

	        END_IF;

	    END_IF;

	END_REGION

	REGION 2 – Activation or deactivation of devices

	    // Change of device state if request is active
	    IF (#sx_OperationReq)                       // Change the device mode twice
	    THEN

	        // Maximum number of Profinet networks
	        #ti_NrOfNetworks := "FC_GetNrOfArrayEl"(iv_Array := #iqa_ProfinetNetworks);

	        // Initial operation request reset
	        #sx_OperationReq := FALSE;

	        // Reset summary error output
	        #qx_Error := FALSE;

	        // A loop operating on Profinet networks
	        FOR #ti_LoopCounterNetworks := 1 TO #ti_NrOfNetworks DO

	            // Maximum number of Profinet devices
	            #ti_NrOfProfinetDevices := "FC_GetNrOfArrayEl"(#iqa_ProfinetNetworks[#ti_LoopCounterNetworks].DeviceStatus);

	            // A loop operating on Profinet devices
	            FOR #ti_LoopCounterDevices := 1 TO ((#ti_NrOfProfinetDevices) - 1) DO

	                // Activation or deactivation device if the device is configured
	                IF (#iqa_ProfinetNetworks[#ti_LoopCounterNetworks].DeviceStatus[#ti_LoopCounterDevices].DeviceState.Configure)                                         // Device configured
	                THEN
	                    // Turning off (mode = 2) or turning on (mode = 1) devices
	                    #si_ActualStatus := D_ACT_DP(REQ := TRUE,
	                                                 MODE := #si_Mode,
	                                                 LADDR := #iqa_ProfinetNetworks[#ti_LoopCounterNetworks].DeviceStatus[#ti_LoopCounterDevices].DeviceState.HW_ID,
	                                                 BUSY => #tx_Busy);

	                    // Operation still required when function "D_ACT_DP" is busy
	                    #sx_OperationReq := #sx_OperationReq OR #tx_Busy;

	                    // Set the output error when D_ACT_DP has an error
	                    IF (INT_TO_WORD(#si_ActualStatus) > 16#8000)    // Error during disabling the devices
	                    THEN

	                        #qx_Error := TRUE;

	                    END_IF;

	                END_IF;

	            END_FOR;

	        END_FOR;

	    END_IF;

	END_REGION

	REGION 3 – Operation done

	    // Update simulation done output
	    #qx_Done := NOT #sx_OperationReq;

	END_REGION
END_FUNCTION_BLOCK

FUNCTION_BLOCK "FB_Loader"
TITLE = FB_Loader
{ S7_Optimized_Access := 'TRUE' }
AUTHOR : MHSE
FAMILY : Equimpent
VERSION : 3.0
// ATTRIBUTES
// AUTO_NUMBER = True
// BLOCK_NUMBER = 216
// END_ATTRIBUTES
//Function block to control loader.
   VAR_INPUT
      iUDT_LoaderConfiguration { ExternalAccessible := 'False'; ExternalVisible := 'False'; ExternalWritable := 'False'} : "UDT_LoaderConfiguration";   //  Loader configuration structure
      ix_SafetyReset { ExternalAccessible := 'False'; ExternalVisible := 'False'; ExternalWritable := 'False'} : Bool;
      ix_SafetyOk { ExternalAccessible := 'False'; ExternalVisible := 'False'; ExternalWritable := 'False'} : Bool;   //  TRUE when Safety Circuit of the Conveyor is healthy
      ix_24vOk { ExternalAccessible := 'False'; ExternalVisible := 'False'; ExternalWritable := 'False'} : Bool;   //  TRUE when 24VDC is healthy
      ix_400vOk { ExternalAccessible := 'False'; ExternalVisible := 'False'; ExternalWritable := 'False'} : Bool;   //  TRUE when 400VAC is healthy
      ix_HardwareOk { ExternalAccessible := 'False'; ExternalVisible := 'False'; ExternalWritable := 'False'} : Bool;   //   TRUE when  hardware is Ok
      ix_ReadyLoad { ExternalAccessible := 'False'; ExternalVisible := 'False'; ExternalWritable := 'False'} : Bool;   //  TRUE when Loader is ready to load
      ix_Running { ExternalAccessible := 'False'; ExternalVisible := 'False'; ExternalWritable := 'False'} : Bool;   //  TRUE when Loader is running
      ix_VFDError { ExternalAccessible := 'False'; ExternalVisible := 'False'; ExternalWritable := 'False'} : Bool;   //  TRUE when Loader has an VFD error
      ix_Healthy { ExternalAccessible := 'False'; ExternalVisible := 'False'; ExternalWritable := 'False'} : Bool;   //  TRUE when Loader has no Errors
      ix_PECEoS { ExternalAccessible := 'False'; ExternalVisible := 'False'; ExternalWritable := 'False'} : Bool;   //  TRUE when the end of section photoeye is not blocked
      ix_PECFull { ExternalAccessible := 'False'; ExternalVisible := 'False'; ExternalWritable := 'False'} : Bool;
      ix_ManualControlled { ExternalAccessible := 'False'; ExternalVisible := 'False'; ExternalWritable := 'False'} : Bool;   //  Loader is manually controlled
      iw_Mode { ExternalAccessible := 'False'; ExternalVisible := 'False'; ExternalWritable := 'False'} : Word;   //  Mode selected on Loader control
      ix_ExternalRequestHold { ExternalAccessible := 'False'; ExternalVisible := 'False'; ExternalWritable := 'False'} : Bool;   //  External request hold
      ix_ResetEnergySave { ExternalAccessible := 'False'; ExternalVisible := 'False'; ExternalWritable := 'False'} : Bool;   //  Reset save energy mode timer
   END_VAR

   VAR_OUTPUT
      qUDT_HMIStatus { ExternalAccessible := 'False'; ExternalVisible := 'False'; ExternalWritable := 'False'} : "UDT_LoaderStatus";   //  HMI status structure
      qUDT_Status { ExternalAccessible := 'False'; ExternalVisible := 'False'; ExternalWritable := 'False'} : "UDT_CommonStatus";   //  Common status structure
      qi_SpeedSelect { ExternalAccessible := 'False'; ExternalVisible := 'False'; ExternalWritable := 'False'} : Int;   //  Speed select (slow, normal or fast)
      qx_EStopReset { ExternalAccessible := 'False'; ExternalVisible := 'False'; ExternalWritable := 'False'} : Bool;
      qx_FaultReset { ExternalAccessible := 'False'; ExternalVisible := 'False'; ExternalWritable := 'False'} : Bool;
      qx_ReleaseLoad { ExternalAccessible := 'False'; ExternalVisible := 'False'; ExternalWritable := 'False'} : Bool;   //  Release Loader
      qx_PECBoS { ExternalAccessible := 'False'; ExternalVisible := 'False'; ExternalWritable := 'False'} : Bool;
   END_VAR

   VAR_IN_OUT
      iqUDT_Statistics : "UDT_LoaderStatistics";   //  Statistics structure
      iqUDT_EquipmentControl : "UDT_EquipmentControl";   //  Equipment control structure
      iqUDT_loaderCommand : "UDT_LoaderCommand";   //  Loader HMI control
      iqUDT_HandShakeUp : "UDT_ConveyorHandshake";   //  Handshake structure
      iqUDT_EquipmentInterface : "UDT_ConveyorInterface";   //  Conveyor interface structure
   END_VAR

   VAR
      sUDT_CommonStatus { ExternalAccessible := 'False'; ExternalVisible := 'False'; ExternalWritable := 'False'; S7_SetPoint := 'False'} : "UDT_CommonStatus";   //  Common status structure
      sUDT_CommonStatusOld { ExternalAccessible := 'False'; ExternalVisible := 'False'; ExternalWritable := 'False'; S7_SetPoint := 'False'} : "UDT_CommonStatus";   //  Auxiliary status structure
      sUDT_HMIStatus { ExternalAccessible := 'False'; ExternalVisible := 'False'; ExternalWritable := 'False'; S7_SetPoint := 'False'} : "UDT_LoaderStatus";   //  HMI status structure
      sFB_PECEoSFiltered { ExternalAccessible := 'False'; ExternalVisible := 'False'; ExternalWritable := 'False'; S7_SetPoint := 'False'} : "FB_TimerOnOffDelay";   //  Filtering end of section photo eye signal
      sFB_EnergySaveTimer { ExternalAccessible := 'False'; ExternalVisible := 'False'; ExternalWritable := 'False'; S7_SetPoint := 'False'} : "FB_TimerOnOffDelay";   //  Timer to start energy save mode
      sFB_CascadeModeTimer { ExternalAccessible := 'False'; ExternalVisible := 'False'; ExternalWritable := 'False'; S7_SetPoint := 'False'} : "FB_TimerOnOffDelay";   //  Timer to cascade start
      sR_TRIG_NotHealthy {InstructionName := 'R_TRIG'; LibVersion := '1.0'; ExternalAccessible := 'False'; ExternalVisible := 'False'; ExternalWritable := 'False'; S7_SetPoint := 'False'} : R_TRIG;   //  Rising edge trigger if extendable not healthy
      sR_TRIG_EnergySave {InstructionName := 'R_TRIG'; LibVersion := '1.0'; ExternalAccessible := 'False'; ExternalVisible := 'False'; ExternalWritable := 'False'; S7_SetPoint := 'False'} : R_TRIG;   //  Rising edge trigger save energy mode active
      sR_TRIG_VFDError {InstructionName := 'R_TRIG'; LibVersion := '1.0'; ExternalAccessible := 'False'; ExternalVisible := 'False'; ExternalWritable := 'False'; S7_SetPoint := 'False'} : R_TRIG;   //  Rising edge of VFD error
      sR_TRIG_ConveyorUp {InstructionName := 'R_TRIG'; LibVersion := '1.0'; ExternalAccessible := 'False'; ExternalVisible := 'False'; ExternalWritable := 'False'; S7_SetPoint := 'False'} : R_TRIG;   //  Rising edge of automatic active
      sR_TRIG_ConveyorDown {InstructionName := 'R_TRIG'; LibVersion := '1.0'; ExternalAccessible := 'False'; ExternalVisible := 'False'; ExternalWritable := 'False'; S7_SetPoint := 'False'} : R_TRIG;   //  Rising edge of automatic not active
      sR_TRIG_StoreMode {InstructionName := 'R_TRIG'; LibVersion := '1.0'; ExternalAccessible := 'False'; ExternalVisible := 'False'; ExternalWritable := 'False'; S7_SetPoint := 'False'} : R_TRIG;   //  Rising edge of extendable in store mode
      sR_TRIG_FeedMode {InstructionName := 'R_TRIG'; LibVersion := '1.0'; ExternalAccessible := 'False'; ExternalVisible := 'False'; ExternalWritable := 'False'; S7_SetPoint := 'False'} : R_TRIG;   //  Rising edge of extendable in feed mode
      sR_TRIG_RunMode {InstructionName := 'R_TRIG'; LibVersion := '1.0'; ExternalAccessible := 'False'; ExternalVisible := 'False'; ExternalWritable := 'False'; S7_SetPoint := 'False'} : R_TRIG;   //  Rising edge of extendable in run mode
      si_AuxEnergySave { ExternalAccessible := 'False'; ExternalVisible := 'False'; ExternalWritable := 'False'} : Int;   //  Auxinalary energy save
      sx_Disabled { ExternalAccessible := 'False'; ExternalVisible := 'False'; ExternalWritable := 'False'} : Bool;   //  Operation is enabled
      sx_PECEoSFiltered { ExternalAccessible := 'False'; ExternalVisible := 'False'; ExternalWritable := 'False'} : Bool;   //  End of section photo eye filtered
      sx_EnergySaveActive { ExternalAccessible := 'False'; ExternalVisible := 'False'; ExternalWritable := 'False'} : Bool;   //  Active energy save mode
      sx_Ready { ExternalAccessible := 'False'; ExternalVisible := 'False'; ExternalWritable := 'False'} : Bool;   //  Conveyor Ready to operate in Automatic mode
      sx_AutomaticActive { ExternalAccessible := 'False'; ExternalVisible := 'False'; ExternalWritable := 'False'} : Bool;   //  Running in automatic
   END_VAR


BEGIN
	(*
	----------------------------------------------------------------------------------------

	Version history:
	Date        | Version   | Author        | Remark
	----------------------------------------------------------------------------------------
	24/05/2019  | 0.1       | F.Baten       | first release MHS TIA 15.1
	17/06/2019  | 0.3       | L.Klar        | Manual mode added to "UDT_EquipmentControl"
	24/07/2019  | 2.0       | L.Klar        | 2.0 MHS library release TIA 15.1
	14/10/2019  | 2.1       | L.Klar        | Updated status structure
	15/10/2019  | 2.2       | S.Deulkar     | Deleted unused symbol, added status
	30/10/2019  | 2.3       | F.Baten       | Pec timer on/off delaytimes interchanged
	04/11/2019  | 2.4       | L.Klar        | First scan bit changed from memory bit to DB variable
	12/11/2019  | 3.0       | P.Majka       | 3.0 MHS library release TIA 15.1
	02/03/2020  | 3.1       | P.Majka       | Adapting reviews
	31/03/2020  | 3.2       | F.Baten       | UDT_UnloaderCommand added
	                                        | Disable by HMI added
	11/01/2021  | 3.3       | L.Klar        | Input safety ok added to stop conveyor condition
	16/02/2021  | 3.4       | K.Pokorski    | HMI Disable fixed
	02/03/2021  | 3.5       | K. Pokorski   | Halted status enable only when automatic on
	15/03/2021  | 3.6       | K. Pokorski   | Energy safe corrected
	21/02/2023  | 4.0       | F.Baten       | 4.0 Release TIA 17.5
	*)

	REGION 1 - Initial

	    REGION 1.1 - First PLC cycle

	        // Bits initialization.
	        IF "DB_Memory".FirstScan
	        THEN
	            #qx_ReleaseLoad := FALSE;
	            #sx_AutomaticActive := FALSE;
	            #iqUDT_HandShakeUp.RTR := FALSE;
	            #iqUDT_HandShakeUp.CascadeStartUp := FALSE;
	            #sx_Disabled := FALSE;
	        END_IF;

	    END_REGION

	    REGION 1.2 Triggers and filters

	        // Rising edge trigger Energy save mode.
	        #sR_TRIG_EnergySave(CLK := #sUDT_CommonStatus.EnergySave);

	        // Rising edge extendable up.
	        #sR_TRIG_ConveyorUp(CLK := #sx_AutomaticActive AND #sx_Ready);

	        // Rising edge extendable down.
	        #sR_TRIG_ConveyorDown(CLK := #sx_AutomaticActive AND NOT #sx_Ready);

	        // Rising edge extendable VFD error.
	        #sR_TRIG_VFDError(CLK := #sUDT_HMIStatus.Specific.VFDError);

	        // Rising edge extendable not healthy .
	        #sR_TRIG_NotHealthy(CLK := #sUDT_HMIStatus.Specific.NotHealthy);

	        // Rising edge extendable feed mode .
	        #sR_TRIG_FeedMode(CLK := #sUDT_HMIStatus.Specific.FeedMode);

	        // Rising edge extendable Store mode .
	        #sR_TRIG_StoreMode(CLK := #sUDT_HMIStatus.Specific.StoreMode);

	        // Rising edge extendable Run mode.
	        #sR_TRIG_RunMode(CLK := #sUDT_HMIStatus.Specific.RunMode);

	        // Filter - End of section photo eye signal filtering.
	        #sFB_PECEoSFiltered(iudi_OnDelayTime := #iUDT_LoaderConfiguration."PEC_EoSTimeOnDelay",
	                            iudi_OffDelayTime := #iUDT_LoaderConfiguration."PEC_EoSTimeOffDelay",
	                            ix_SignalToDelay := #ix_PECEoS,
	                            ix_Enable := #ix_Running,
	                            qx_DelayedSignal => #sx_PECEoSFiltered);

	    END_REGION

	    REGION HMI button Disable/Enable operation
	        IF #iqUDT_loaderCommand.Disable
	        THEN
	            #sx_Disabled := TRUE;
	        ELSE
	            #sx_Disabled := FALSE;
	        END_IF;
	        #iqUDT_loaderCommand.Disable := FALSE;

	        // Copy status to HMI
	        #sUDT_HMIStatus.Specific.Disabled := #sx_Disabled;

	    END_REGION
	END_REGION

	REGION 2 - Errors

	    // VFD Error.
	    #sUDT_HMIStatus.Specific.VFDError := (#ix_VFDError AND #ix_400vOk AND #ix_HardwareOk);

	    // Not healthy.
	    #sUDT_HMIStatus.Specific.NotHealthy := (NOT #ix_Healthy AND #ix_400vOk AND #ix_24vOk AND #ix_HardwareOk);

	    // Common Error.
	    #sUDT_CommonStatus.Error := NOT #ix_24vOk
	    OR NOT #ix_400vOk
	    OR NOT #ix_HardwareOk
	    OR NOT #ix_SafetyOk
	    OR #sUDT_HMIStatus.Specific.VFDError
	    OR #sUDT_HMIStatus.Specific.NotHealthy;

	    // Warning.
	    #sUDT_CommonStatus.Warning := FALSE;

	    // Mode selected = 1.
	    IF #iw_Mode = 1
	    THEN
	        #sUDT_HMIStatus.Specific.StoreMode := TRUE;
	        #sUDT_HMIStatus.Specific.FeedMode := FALSE;
	        #sUDT_HMIStatus.Specific.RunMode := FALSE;
	    END_IF;

	    // Mode selected = 2.
	    IF #iw_Mode = 2
	    THEN
	        #sUDT_HMIStatus.Specific.StoreMode := FALSE;
	        #sUDT_HMIStatus.Specific.FeedMode := TRUE;
	        #sUDT_HMIStatus.Specific.RunMode := FALSE;
	    END_IF;

	    // Mode selected = 3.
	    IF #iw_Mode = 3
	    THEN
	        #sUDT_HMIStatus.Specific.StoreMode := FALSE;
	        #sUDT_HMIStatus.Specific.FeedMode := FALSE;
	        #sUDT_HMIStatus.Specific.RunMode := TRUE;
	    END_IF;

	END_REGION

	REGION 3 - Check conditions to set loader ready

	    // Ready to operate.
	    #sx_Ready := NOT #sUDT_CommonStatus.Error
	    AND #ix_Healthy
	    AND NOT #ix_ManualControlled;

	END_REGION

	REGION 4 - Stop loader

	    // Reset bits to stop loader.
	    IF NOT #iqUDT_EquipmentControl.Command.AutomaticOn
	        OR #sUDT_CommonStatus.Error
	        OR #ix_ManualControlled
	    THEN
	        #sx_AutomaticActive := FALSE;
	        #iqUDT_HandShakeUp.RTR := FALSE;
	        #iqUDT_HandShakeUp.CascadeStartUp := FALSE;
	    END_IF;

	END_REGION

	REGION 5 - Start Automatic mode

	    REGION 5.1 - Start

	        // Activating automatic mode.
	        IF #iqUDT_EquipmentControl.Command.Start
	            AND #sx_Ready
	        THEN
	            #sx_AutomaticActive := TRUE;
	        END_IF;

	    END_REGION

	    REGION 5.2 - Cascade mode

	        // Timer to cascade mode.
	        #sFB_CascadeModeTimer(iudi_OnDelayTime := #iUDT_LoaderConfiguration.CascadeTimeOnDelay,
	                              ix_SignalToDelay := #sx_AutomaticActive,
	                              ix_Enable := NOT #iqUDT_HandShakeUp.CascadeStartUp,
	                              qx_DelayedSignal => #iqUDT_HandShakeUp.CascadeStartUp);

	    END_REGION

	END_REGION

	REGION 6 - Automatic mode active

	    REGION 6.1 - Operation

	        // Run/release load: starting and stopping is controlled by loader controls.
	        #qx_ReleaseLoad := #sx_AutomaticActive
	        AND #sx_Ready
	        AND #ix_ReadyLoad
	        AND NOT #sx_Disabled
	        AND NOT #ix_ExternalRequestHold
	        AND NOT #sx_EnergySaveActive;

	        // Ready to receive.
	        #iqUDT_HandShakeUp.RTR := #sx_AutomaticActive
	        AND #sx_Ready
	        AND #ix_ReadyLoad
	        AND NOT #ix_ExternalRequestHold;

	    END_REGION

	    REGION 6.2 - Energy save
	        IF #iUDT_LoaderConfiguration.Energy THEN

	            // Set Energy save active.
	            IF #si_AuxEnergySave >= #iUDT_LoaderConfiguration.EnergySaveLength
	            THEN
	                #sx_EnergySaveActive := TRUE;
	            END_IF;

	            // Reset or increment displacement calculation to use for energy save.
	            IF (NOT #sx_PECEoSFiltered
	                OR #iqUDT_HandShakeUp.RTS
	                OR #iqUDT_HandShakeUp.ResetEnergySave
	                OR #ix_ResetEnergySave
	                OR #ix_ManualControlled
	                OR NOT #ix_ReadyLoad)
	            THEN
	                #si_AuxEnergySave := 0;
	                #sx_EnergySaveActive := FALSE;
	            ELSE
	                #si_AuxEnergySave += #iqUDT_EquipmentInterface.Displacement;
	            END_IF;

	        ELSE

	            #si_AuxEnergySave := 0;
	            #sx_EnergySaveActive := FALSE;

	        END_IF;
	    END_REGION

	END_REGION

	REGION 7 - Speed control

	    // Copy speed setpoint from configuration.
	    #qi_SpeedSelect := #iUDT_LoaderConfiguration.Speedsetpoint;

	    // Clear speed setpoint depending on wrong configuration.
	    IF #iUDT_LoaderConfiguration.Speedsetpoint < 0
	        OR #iUDT_LoaderConfiguration.Speedsetpoint > 2
	    THEN
	        #qi_SpeedSelect := 0;
	    END_IF;

	END_REGION

	REGION 8 - Reset
	    // Fault and Estop reset outputs
	    #qx_FaultReset := #ix_SafetyReset OR #iqUDT_EquipmentControl.Command.Reset;
	    #qx_EStopReset := #ix_SafetyReset;

	END_REGION

	REGION 9 Output enable

	    #qx_PECBoS := #ix_PECFull;

	END_REGION

	REGION 10 - Statistics

	    // Up Time.
	    IF #sx_AutomaticActive
	        AND #sx_Ready
	        OR #iqUDT_EquipmentControl.Command.ResetData
	    THEN
	        "FC_Statistics"(ix_Reset := #iqUDT_EquipmentControl.Command.ResetData,
	                        ix_Activate := #sx_AutomaticActive AND #sx_Ready,
	                        ix_RTrigActivate := #sR_TRIG_ConveyorUp.Q,
	                        iqUDT_Statistics := #iqUDT_Statistics.ExtendableUpTime);
	    END_IF;

	    // Down Time.
	    IF #sx_AutomaticActive
	        AND #sx_Ready
	        OR #iqUDT_EquipmentControl.Command.ResetData
	    THEN
	        "FC_Statistics"(ix_Reset := #iqUDT_EquipmentControl.Command.ResetData,
	                        ix_Activate := #sx_AutomaticActive AND NOT #sx_Ready,
	                        ix_RTrigActivate := #sR_TRIG_ConveyorDown.Q,
	                        iqUDT_Statistics := #iqUDT_Statistics.ExtendableDownTime);
	    END_IF;

	    // Energy save mode active.
	    IF #sx_EnergySaveActive
	        OR #iqUDT_EquipmentControl.Command.ResetData
	    THEN
	        "FC_Statistics"(ix_Reset := #iqUDT_EquipmentControl.Command.ResetData,
	                        ix_Activate := #sUDT_CommonStatus.EnergySave,
	                        ix_RTrigActivate := #sR_TRIG_EnergySave.Q,
	                        iqUDT_Statistics := #iqUDT_Statistics.EnergySave);
	    END_IF;

	    // VFD Error.
	    IF #sUDT_HMIStatus.Specific.VFDError
	        OR #iqUDT_EquipmentControl.Command.ResetData
	    THEN
	        "FC_Statistics"(ix_Reset := #iqUDT_EquipmentControl.Command.ResetData,
	                        ix_Activate := #sUDT_HMIStatus.Specific.VFDError,
	                        ix_RTrigActivate := #sR_TRIG_VFDError.Q,
	                        iqUDT_Statistics := #iqUDT_Statistics.VFDError);
	    END_IF;

	    // Not healthy.
	    IF #sUDT_HMIStatus.Specific.NotHealthy
	        OR #iqUDT_EquipmentControl.Command.ResetData
	    THEN
	        "FC_Statistics"(ix_Reset := #iqUDT_EquipmentControl.Command.ResetData,
	                        ix_Activate := #sUDT_HMIStatus.Specific.NotHealthy,
	                        ix_RTrigActivate := #sR_TRIG_NotHealthy.Q,
	                        iqUDT_Statistics := #iqUDT_Statistics.NotHealthy);
	    END_IF;

	END_REGION

	REGION 11 - Status

	    // Set statuses.
	    #sUDT_CommonStatus.Stopped := NOT #sx_AutomaticActive;
	    #sUDT_CommonStatus.Running := #ix_Running;
	    #sUDT_CommonStatus.AutoON := #sx_Ready AND #sx_AutomaticActive;
	    #sUDT_CommonStatus.Halted := #ix_ExternalRequestHold AND #sUDT_CommonStatus.AutoON;
	    #sUDT_CommonStatus.Manual := #ix_ManualControlled;
	    #sUDT_CommonStatus.ManualRun := #sUDT_CommonStatus.Manual AND #sUDT_CommonStatus.Running;
	    #sUDT_CommonStatus.EnergySave := #sx_EnergySaveActive;
	    #sUDT_CommonStatus.SafetyStop := NOT #ix_SafetyOk;


	    // HMI status update on change.
	    IF #sUDT_CommonStatusOld <> #sUDT_CommonStatus
	        OR (#sR_TRIG_FeedMode.Q OR #sR_TRIG_StoreMode.Q OR #sR_TRIG_RunMode.Q)
	    THEN
	        // HMI status initialization.
	        #sUDT_HMIStatus.Status := 0;

	        // Energy save.
	        IF #sUDT_CommonStatus.EnergySave
	        THEN
	            #sUDT_HMIStatus.Status := "DB_HMIStatusConfiguration".EnergySave;
	        END_IF;

	        // Running.
	        IF #sUDT_CommonStatus.Running
	        THEN
	            #sUDT_HMIStatus.Status := "DB_HMIStatusConfiguration".Running;
	        END_IF;

	        // Stopped.
	        IF #sUDT_CommonStatus.Stopped
	        THEN
	            #sUDT_HMIStatus.Status := "DB_HMIStatusConfiguration".Stopped;
	        END_IF;

	        // Dieback.
	        IF #sUDT_CommonStatus.Dieback
	        THEN
	            #sUDT_HMIStatus.Status := "DB_HMIStatusConfiguration".Dieback;
	        END_IF;

	        // Halted.
	        IF #sUDT_CommonStatus.Halted
	        THEN
	            #sUDT_HMIStatus.Status := "DB_HMIStatusConfiguration".Halted;
	        END_IF;

	        // Manual.
	        IF #sUDT_CommonStatus.Manual
	        THEN
	            #sUDT_HMIStatus.Status := "DB_HMIStatusConfiguration".Manual;
	        END_IF;

	        // Running in manual mode.
	        IF #sUDT_CommonStatus.ManualRun
	        THEN
	            #sUDT_HMIStatus.Status := "DB_HMIStatusConfiguration".ManualRun;
	        END_IF;

	        // Not healthy.
	        IF #sUDT_HMIStatus.Specific.NotHealthy
	        THEN
	            #sUDT_HMIStatus.Status := "DB_HMIStatusConfiguration".VFDNotHealthy;
	        END_IF;

	        // VFD error.
	        IF #sUDT_HMIStatus.Specific.VFDError
	        THEN
	            #sUDT_HMIStatus.Status := "DB_HMIStatusConfiguration".VFDError;
	        END_IF;

	        // Safety stop.
	        IF (#sUDT_CommonStatus.SafetyStop)
	        THEN
	            #sUDT_HMIStatus.Status := "DB_HMIStatusConfiguration".SafetyStop;
	        END_IF;

	        // Copy statuses.

	        #sUDT_CommonStatusOld := #sUDT_CommonStatus;

	    END_IF;
	    #qUDT_HMIStatus := #sUDT_HMIStatus;
	    #qUDT_Status := #sUDT_CommonStatus;

	END_REGION

	REGION 11 - Report to control block

	    "FC_EquipmentReport"(iUDT_Status := #sUDT_CommonStatus,
	                         iqUDT_Control := #iqUDT_EquipmentControl);

	END_REGION
END_FUNCTION_BLOCK

FUNCTION_BLOCK "FB_PECUpdateD"
TITLE = FB_PECUpdate
{ S7_Optimized_Access := 'TRUE' }
AUTHOR : MHSE
FAMILY : GeneralSystemFunctions
VERSION : 3.0
// ATTRIBUTES
// AUTO_NUMBER = True
// BLOCK_NUMBER = 23
// END_ATTRIBUTES
//Function block to update parcel data in a tracking array at PEC position.
   VAR_INPUT
      iUDT_PECUpdateConfiguration { ExternalAccessible := 'False'; ExternalVisible := 'False'; ExternalWritable := 'False'} : "UDT_PECDUpdateConfiguration";   //   PEC update configuration
      iUDT_ConveyorCommonConfiguration { ExternalAccessible := 'False'; ExternalVisible := 'False'; ExternalWritable := 'False'} : "UDT_ConveyorCommonConfiguration";   //   Conveyor configuration
      ix_PEC { ExternalAccessible := 'False'; ExternalVisible := 'False'; ExternalWritable := 'False'} : Bool;   //   TRUE when the end of section photoeye is not blocked
      ix_TeachingMode { ExternalAccessible := 'False'; ExternalVisible := 'False'; ExternalWritable := 'False'} : Bool;   //   Teaching mode enable
   END_VAR

   VAR_OUTPUT
      qUDT_Status { ExternalAccessible := 'False'; ExternalVisible := 'False'; ExternalWritable := 'False'} : "UDT_PECUpdateStatus";   //   Status structure
      qi_GINwrite { ExternalAccessible := 'False'; ExternalVisible := 'False'; ExternalWritable := 'False'} : Int;   //  Gin found or generated
      qx_PECFiltered { ExternalAccessible := 'False'; ExternalVisible := 'False'; ExternalWritable := 'False'} : Bool;   //   Filtered photoeye signal
   END_VAR

   VAR_IN_OUT
      iqa_TrackingData : Array[*] of Int;   //   Tracking data
      iqUDT_ConveyorInterface : "UDT_ConveyorInterface";   //   Conveyor interface
      iqUDT_UnknownGINRange : "UDT_UnknownGIN";   //   Unknown GIN
      iqUDT_FifoHeader : "UDT_FifoHeader";   //   FIFO header
      iqa_FifoData : Array[*] of Int;   //   FIFO data
      iqUDT_Statistics : "UDT_PECUpdateStatistics";   //   Statistic structure
   END_VAR

   VAR
      sFB_PEC { ExternalAccessible := 'False'; ExternalVisible := 'False'; ExternalWritable := 'False'; S7_SetPoint := 'False'} : "FB_PECD";   //   Photoeye function
      sFB_LengthMeasurement { ExternalAccessible := 'False'; ExternalVisible := 'False'; ExternalWritable := 'False'; S7_SetPoint := 'False'} : "FB_ParcelLength";   //   Length measurement
      s_R_TRIG_Parcel {InstructionName := 'R_TRIG'; LibVersion := '1.0'; ExternalAccessible := 'False'; ExternalVisible := 'False'; ExternalWritable := 'False'; S7_SetPoint := 'False'} : R_TRIG;   //   Parcel detected rising edge to count parcels
      s_R_TRIG_ParcelFound {InstructionName := 'R_TRIG'; LibVersion := '1.0'; ExternalAccessible := 'False'; ExternalVisible := 'False'; ExternalWritable := 'False'; S7_SetPoint := 'False'} : R_TRIG;   //   Parcel detected rising edge to update the PEC position tracking record
      s_R_TRIG_DataFound {InstructionName := 'R_TRIG'; LibVersion := '1.0'; ExternalAccessible := 'False'; ExternalVisible := 'False'; ExternalWritable := 'False'; S7_SetPoint := 'False'} : R_TRIG;   //   Any data found at a PEC position rising edge
      s_R_TRIG_PositiveDataFound {InstructionName := 'R_TRIG'; LibVersion := '1.0'; ExternalAccessible := 'False'; ExternalVisible := 'False'; ExternalWritable := 'False'; S7_SetPoint := 'False'} : R_TRIG;   //   Positive data found at a PEC position rising edge
      s_R_TRIG_TeachMode {InstructionName := 'R_TRIG'; LibVersion := '1.0'; ExternalAccessible := 'False'; ExternalVisible := 'False'; ExternalWritable := 'False'; S7_SetPoint := 'False'} : R_TRIG;   //   Teaching mode activation rising edge
      s_R_TRIG_TooManyLost {InstructionName := 'R_TRIG'; LibVersion := '1.0'; ExternalAccessible := 'False'; ExternalVisible := 'False'; ExternalWritable := 'False'; S7_SetPoint := 'False'} : R_TRIG;   //   Too many lost parcels error statistics trigger
      sUDT_LostGINFIFOStatus { ExternalAccessible := 'False'; ExternalVisible := 'False'; ExternalWritable := 'False'; S7_SetPoint := 'False'} : "UDT_FifoStatus";   //   Lost GIN FIFO status
      "ss_PEC/DataDeviation" { ExternalAccessible := 'False'; ExternalVisible := 'False'; ExternalWritable := 'False'} : Struct   // PEC/Data deviation calculation structure
         "Type" { ExternalAccessible := 'False'; ExternalVisible := 'False'; ExternalWritable := 'False'} : Int;   // 1= match, 2 = PEC no Data, 3= Data no PEC, 4 Double data, 5 = Pec no data Lost
         Last { ExternalAccessible := 'False'; ExternalVisible := 'False'; ExternalWritable := 'False'} : Int;   //  Last deviation of found data [cm]
         GIN { ExternalAccessible := 'False'; ExternalVisible := 'False'; ExternalWritable := 'False'} : Int;   //  Last GIN deviation
         Sum { ExternalAccessible := 'False'; ExternalVisible := 'False'; ExternalWritable := 'False'} : Int;   //  Deviation sum [cm]
         Nr { ExternalAccessible := 'False'; ExternalVisible := 'False'; ExternalWritable := 'False'} : Int;   //  Deviation number
      END_STRUCT;
      ss_ValidGINRange { ExternalAccessible := 'False'; ExternalVisible := 'False'; ExternalWritable := 'False'} : Struct   //   Valid GIN range
         Start { ExternalAccessible := 'False'; ExternalVisible := 'False'; ExternalWritable := 'False'} : Int;
         End { ExternalAccessible := 'False'; ExternalVisible := 'False'; ExternalWritable := 'False'} : Int;
         GIN { ExternalAccessible := 'False'; ExternalVisible := 'False'; ExternalWritable := 'False'} : Int;
      END_STRUCT;
      ss_AlignedParcelsCounters { ExternalAccessible := 'False'; ExternalVisible := 'False'; ExternalWritable := 'False'} : Struct   //   Aligned parcels counters
         Total { ExternalAccessible := 'False'; ExternalVisible := 'False'; ExternalWritable := 'False'} : Int;   //   Total aligned parcels
         DataNoPEC { ExternalAccessible := 'False'; ExternalVisible := 'False'; ExternalWritable := 'False'} : Int;   //   Parcels aligned in case data detected without photoeye signal
         PECNoData { ExternalAccessible := 'False'; ExternalVisible := 'False'; ExternalWritable := 'False'} : Int;   //   Parcels aligned in case parcel detected without data
      END_STRUCT;
      ss_LostParcelsCounters { ExternalAccessible := 'False'; ExternalVisible := 'False'; ExternalWritable := 'False'} : Struct   //   Lost parcels counters
         Total { ExternalAccessible := 'False'; ExternalVisible := 'False'; ExternalWritable := 'False'} : Int;   //   Total number of lost parcels
         DoubleData { ExternalAccessible := 'False'; ExternalVisible := 'False'; ExternalWritable := 'False'} : Int;   //   Parcels lost due to double data found in a search window
         ParcelNotFound { ExternalAccessible := 'False'; ExternalVisible := 'False'; ExternalWritable := 'False'} : Int;   //   Parcels lost due to no parcel detected after travelling search window distance
      END_STRUCT;
      ss_LostValidParcelsCounters { ExternalAccessible := 'False'; ExternalVisible := 'False'; ExternalWritable := 'False'} : Struct   //   Lost parcels counters
         Total { ExternalAccessible := 'False'; ExternalVisible := 'False'; ExternalWritable := 'False'} : Int;   //   Total number of lost parcels
         DoubleData { ExternalAccessible := 'False'; ExternalVisible := 'False'; ExternalWritable := 'False'} : Int;   //   Parcels lost due to double data found in a search window
         ParcelNotFound { ExternalAccessible := 'False'; ExternalVisible := 'False'; ExternalWritable := 'False'} : Int;   //   Parcels lost due to no parcel detected after travelling search window distance
      END_STRUCT;
      si_UnknownParcelsCounters { ExternalAccessible := 'False'; ExternalVisible := 'False'; ExternalWritable := 'False'} : Struct   //   Unknown parcels counters
         Total { ExternalAccessible := 'False'; ExternalVisible := 'False'; ExternalWritable := 'False'} : Int;   //   Total number of unknown parcels
         LostParcelFound { ExternalAccessible := 'False'; ExternalVisible := 'False'; ExternalWritable := 'False'} : Int;   //   Parcel found with a lost data, unknown GIN created
         DataNotFound { ExternalAccessible := 'False'; ExternalVisible := 'False'; ExternalWritable := 'False'} : Int;   //   Data not found during search window scan
      END_STRUCT;
      slr_Performance { ExternalAccessible := 'False'; ExternalVisible := 'False'; ExternalWritable := 'False'} : LReal := 100.0;   //   Update performance [%]
      sdi_TotalNumberOfParcels { ExternalAccessible := 'False'; ExternalVisible := 'False'; ExternalWritable := 'False'} : DInt;   //   Total number of parcels detected
      sdi_TotalNumberOfData { ExternalAccessible := 'False'; ExternalVisible := 'False'; ExternalWritable := 'False'} : DInt;   //   Total number of data detected
      si_PECPosition { ExternalAccessible := 'False'; ExternalVisible := 'False'; ExternalWritable := 'False'} : Int;   //   Photoeye position [cm]
      si_SearchWindow { ExternalAccessible := 'False'; ExternalVisible := 'False'; ExternalWritable := 'False'} : Int;   //   Data search distance from photoeye position [cm]
      si_GINToWrite { ExternalAccessible := 'False'; ExternalVisible := 'False'; ExternalWritable := 'False'} : Int;   //   Found or generated GIN, which will be used to update photoeye position in the tracking array
      si_PositionToUpdate { ExternalAccessible := 'False'; ExternalVisible := 'False'; ExternalWritable := 'False'} : Int;   //   Position in a tracking array to be updated
      si_Direction { ExternalAccessible := 'False'; ExternalVisible := 'False'; ExternalWritable := 'False'} : Int;   //   Direction of the displacement to parametrize loops
      si_Displacement { ExternalAccessible := 'False'; ExternalVisible := 'False'; ExternalWritable := 'False'} : Int;   //   Displacement [cm]
      si_ParcelWaitDistance { ExternalAccessible := 'False'; ExternalVisible := 'False'; ExternalWritable := 'False'} : Int;   //   Parcel delay [cm]
      si_LastUpdatedGIN { ExternalAccessible := 'False'; ExternalVisible := 'False'; ExternalWritable := 'False'} : Int;   //   Last updated GIN to check if next data is a new one
      si_LastCountedData { ExternalAccessible := 'False'; ExternalVisible := 'False'; ExternalWritable := 'False'} : Int;   //   Last counted data
      si_LostParcelsInARow { ExternalAccessible := 'False'; ExternalVisible := 'False'; ExternalWritable := 'False'} : Int;   //   Number of lost parcel in a row
      si_NumberOfTeachedParcels { ExternalAccessible := 'False'; ExternalVisible := 'False'; ExternalWritable := 'False'} : Int;   //   Number of teached parcels
      si_AverageSlip { ExternalAccessible := 'False'; ExternalVisible := 'False'; ExternalWritable := 'False'} : Int;   //   Average parcel slip [cm]
      si_CalculatedLengthCorrection { ExternalAccessible := 'False'; ExternalVisible := 'False'; ExternalWritable := 'False'} : Int;   //   Calculated length correction after teaching
      si_ParcelLengthFilterCounter { ExternalAccessible := 'False'; ExternalVisible := 'False'; ExternalWritable := 'False'} : Int;   //  Parcel length filter counter [cm]
      si_ParcelLengthFilterOldGIN { ExternalAccessible := 'False'; ExternalVisible := 'False'; ExternalWritable := 'False'} : Int;   //  Parcel length filter old GIN
      si_i { ExternalAccessible := 'False'; ExternalVisible := 'False'; ExternalWritable := 'False'} : Int;   //   Loop counter
      sx_ParcelDetected { ExternalAccessible := 'False'; ExternalVisible := 'False'; ExternalWritable := 'False'} : Bool;   //   Parcel detected
      sx_ParcelWaitEnable { ExternalAccessible := 'False'; ExternalVisible := 'False'; ExternalWritable := 'False'} : Bool;   //   Missing parcel monitoring
      sx_TeachingMode { ExternalAccessible := 'False'; ExternalVisible := 'False'; ExternalWritable := 'False'} : Bool;   //   Teaching mode
      sx_GenerateGIN { ExternalAccessible := 'False'; ExternalVisible := 'False'; ExternalWritable := 'False'} : Bool;   //   Request to generate GIN
      sx_LostGINFIFOError { ExternalAccessible := 'False'; ExternalVisible := 'False'; ExternalWritable := 'False'} : Bool;   //   Lost GIN FIFO error
      sx_LostGINFIFOWarning { ExternalAccessible := 'False'; ExternalVisible := 'False'; ExternalWritable := 'False'} : Bool;   //   Lost GIN FIFO warning
      sx_InvalidDirection { ExternalAccessible := 'False'; ExternalVisible := 'False'; ExternalWritable := 'False'} : Bool;   //   Invalid direction
      sx_InvalidGINRange { ExternalAccessible := 'False'; ExternalVisible := 'False'; ExternalWritable := 'False'} : Bool;   //   Invalid GIN range
      sx_InvalidDisplacement { ExternalAccessible := 'False'; ExternalVisible := 'False'; ExternalWritable := 'False'} : Bool;   //   Invalid displacement
      sx_InvalidSearchWindow { ExternalAccessible := 'False'; ExternalVisible := 'False'; ExternalWritable := 'False'} : Bool;   //   Invalid search window
      sx_DoubleDataFound { ExternalAccessible := 'False'; ExternalVisible := 'False'; ExternalWritable := 'False'} : Bool;   //   Double data detected
      sx_LengthMeasurementEnable { ExternalAccessible := 'False'; ExternalVisible := 'False'; ExternalWritable := 'False'} : Bool;
   END_VAR

   VAR_TEMP
      tUDT_PECConfiguration : "UDT_PECDConfiguration";   //   PEC configuration
      tUDT_PECStatus : "UDT_PECStatus";   //   PEC status
   END_VAR

   VAR CONSTANT
      ci_ZeroGIN : Int;   //   GIN = 0
   END_VAR


BEGIN
	(*
	----------------------------------------------------------------------------------------

	Version history:
	Date        | Version   | Author        | Remark
	----------------------------------------------------------------------------------------
	24/05/2019  | 0.1       | L.Klar        | first release MHSE TIA 15.1
	13/06/2019  | 0.2       | A.Nowak       | Replacement of instruction if for direct write into variable
	21/06/2019  | 0.3       | A.Nowak       | Add gap mesurement function and reorganise block (regions)
	24/07/2019  | 2.0       | L.Klar        | 2.0 MHSE library release TIA 15.1
	23/08/2019  | 2.1       | L.Klar        | "UDT_ConveyorConfiguration" changed to "UDT_ConveyorCommonConfiguration"
	XX/08/2019  | 2.2       | L.Klar        | Update logic changed
	19/09/2019  | 2.3       | P.Majka       | Updating checking PEC and PEC filtered signals
	30/09/2019  | 2.4       | L.Klar        | FB_PEC added, Filtered PEC signal output added
	21/10/2019  | 2.6       | L.Klar        | Configuration UDT chanaged to input, PEC configuration interface input name changed
	23/10/2019  | 2.7       | P.Majka       | Added Region 1, renumerating Regions, changed logic in Region 10.3 and Region 5
	29/10/2019  | 2.8       | L.Klar        | FB_PEC call changed
	14/11/2019  | 2.9       | L.Klar        | Deviations calculation corrected
	14/11/2019  | 3.0       | P.Majka       | 3.0 MHSE library release TIA 15.1
	20/12/2019  | 3.1       | S.Deulkar     | Used configureation error bit to report to conveyor block
	07/01/2020  | 3.2       | L.Klar        | GIN record structure updated, GIN cleared with default one during generation
	                                        | PECUpdate configuration UDT update - search window DINT -> INT,
	                                        | Conveyor common configuration UDT update - length INT -> DINT  conversion added
	29/01/2020  | 3.3       | L.Klar        | Negative GIN handling fixed, configuration bit added to delete negative GIN instead of ignoing it.
	24/02/2020  | 3.4       | L.Klar        | Formating changes, statistics counter added
	10/03/2020  | 3.5       | F.Baten       | Range check unknown GIN region 7
	26/03/2020  | 3.6       | F.Baten       | Added output 'qi_GINwrite'
	25/11/2020  | 3.7       | L.Klar        | Length filter added
	07/12/2020  | 3.8       | L.Klar        | Length filter bug fix
	22/01/2021  | 3.9       | L.Klar        | Total number of parcels and lost parcels counter fixed
	14/08/2021  | 3.10      | S. Deulkar    | Update from EMA
	20/04/2023  | 4.0       | F.Baten       | Added deviation parameter for easier configuration
	                                        | PEC delay changed to distance
	                                        | 4.0 Release TIA 17.5
	*)



	REGION 1 – FIFO header status update

	    "FC_Fifo"(ic_Mode := 'S',
	              qUDT_Status => #sUDT_LostGINFIFOStatus,
	              qx_Error => #sx_LostGINFIFOError,
	              qx_Warning => #sx_LostGINFIFOWarning,
	              iqv_Data := #si_GINToWrite,
	              iqUDT_FifoHeader := #iqUDT_FifoHeader,
	              iqv_DataBuffer := #iqa_FifoData);

	END_REGION

	REGION 2 – Displacement read

	    #si_Displacement := #iqUDT_ConveyorInterface.Displacement;

	END_REGION

	REGION 3 – PEC Position conversion from mm to cm

	    // The conversion is required because the photoeye position is given in mm and the tracking resolution is 1 cm.
	    #si_PECPosition := DINT_TO_INT(#iUDT_PECUpdateConfiguration.Distance / 10);

	END_REGION

	REGION 4 – Teaching mode enable

	    (* Teaching mode is used to calculate conveyor length correction, which allows to align real conveyor length with a tracking array length.
	       Correction is calculated as a difference between photoeye signal and tracking data deviations.
	       Calculated correction has to be manually copied from a FB_PECUpdate instance data block to conveyor configuration.*)

	    // Teaching mode is initialized and activated manually via block input.
	    #s_R_TRIG_TeachMode(CLK := #ix_TeachingMode);

	    IF (#s_R_TRIG_TeachMode.Q
	        AND NOT #sx_TeachingMode)
	    THEN
	        #"ss_PEC/DataDeviation".Type := 0;
	        #"ss_PEC/DataDeviation".Nr := 0;
	        #"ss_PEC/DataDeviation".Sum := 0;
	        #si_NumberOfTeachedParcels := 0;
	        #sx_TeachingMode := TRUE;
	    END_IF;

	END_REGION

	REGION 5 – Photoeye

	    (*FB_PEC block call to filter photoeye signal and calculate jam status.*)

	    // Copy PEC configuration.
	    #tUDT_PECConfiguration.Distance := #iUDT_PECUpdateConfiguration.Distance;
	    #tUDT_PECConfiguration.JamDisplacementLimit := #iUDT_PECUpdateConfiguration.JamDisplacementLimit;
	    #tUDT_PECConfiguration.OnDelayDistance := #iUDT_PECUpdateConfiguration.OnDelayDistance;
	    #tUDT_PECConfiguration.OffDelayDistance := #iUDT_PECUpdateConfiguration.OffDelayDistance;
	    #tUDT_PECConfiguration.ResetWithPECBlocked := #iUDT_PECUpdateConfiguration.ResetWithPECBlocked;

	    //Call FB_PEC.
	    #sFB_PEC(ix_PEC := #ix_PEC,
	             iUDT_PECConfiguration := #tUDT_PECConfiguration,
	             qUDT_HMIStatus => #tUDT_PECStatus,
	             iqUDT_ConveyorInterface := #iqUDT_ConveyorInterface,
	             iqUDT_PECStatistics := #iqUDT_Statistics.PEC);

	    // Parcel length filter
	    IF NOT #ix_PEC
	        AND #iUDT_PECUpdateConfiguration.ParcelLengthFilter
	        AND #iqa_TrackingData[#si_PECPosition - 1] > 0
	        AND #iqa_TrackingData[#si_PECPosition - 1] <> #si_ParcelLengthFilterOldGIN THEN

	        IF "DB_GIN".GIN[#iqa_TrackingData[#si_PECPosition - 1]].General.Length > 0 THEN
	            #si_ParcelLengthFilterCounter := "DB_GIN".GIN[#iqa_TrackingData[#si_PECPosition - 1]].General.Length;
	        END_IF;

	        #si_ParcelLengthFilterOldGIN := #iqa_TrackingData[#si_PECPosition - 1];

	    END_IF;

	    IF #si_ParcelLengthFilterCounter > 0 THEN

	        #qUDT_Status.PEC := FALSE;
	        #qx_PECFiltered := FALSE;
	        #si_ParcelLengthFilterCounter -= #iqUDT_ConveyorInterface.Displacement;

	    ELSE

	        #qUDT_Status.PEC := #sFB_PEC.qx_PECFiltered;
	        #qx_PECFiltered := #sFB_PEC.qx_PECFiltered;

	    END_IF;

	    #qUDT_Status.Jam := #tUDT_PECStatus.Jam;

	    // Parcel detected variable to simplify further photoeye position tracking record update.
	    #sx_ParcelDetected := NOT #qUDT_Status.PEC;

	END_REGION

	REGION 6 – Error reset

	    // Reset errors when reset signal is given.
	    IF (#iqUDT_ConveyorInterface.InternalErrorReset)
	    THEN
	        #si_LostParcelsInARow := 0;
	        #qUDT_Status.TooManyLost := FALSE;
	        #sx_InvalidDisplacement := FALSE;
	    END_IF;

	END_REGION

	REGION 7 – GIN generator initialization

	    // Valid GIN range configuration is moved to a structure.
	    #ss_ValidGINRange.Start := #iUDT_PECUpdateConfiguration.GINRangeStart;
	    #ss_ValidGINRange.End := #iUDT_PECUpdateConfiguration.GINRangeEnd;

	    // Check if the unknown GIN is within range
	    IF #iqUDT_UnknownGINRange.GIN < #iqUDT_UnknownGINRange.Start
	        OR #iqUDT_UnknownGINRange.GIN > #iqUDT_UnknownGINRange.End
	    THEN
	        #iqUDT_UnknownGINRange.GIN := #iqUDT_UnknownGINRange.Start;
	    END_IF;

	    // Whenever valid GIN range is changed and the generated GIN doesn't fit, it's initialized.
	    IF (#ss_ValidGINRange.GIN < #ss_ValidGINRange.Start
	        OR #ss_ValidGINRange.GIN > #ss_ValidGINRange.End)
	    THEN
	        #ss_ValidGINRange.GIN := #ss_ValidGINRange.Start;
	    END_IF;

	    // Valid GIN range is set locally in PEC update configuration structure and it can't overlap with a global unknown GIN range.
	    #sx_InvalidGINRange := #iUDT_PECUpdateConfiguration.GenerationPoint
	    AND (#ss_ValidGINRange.End <= #ss_ValidGINRange.Start
	    OR #ss_ValidGINRange.Start <= #iqUDT_UnknownGINRange.End
	    OR #iqUDT_UnknownGINRange.End <= #iqUDT_UnknownGINRange.Start)
	    AND #ss_ValidGINRange.Start < 1000;   // Until 1000 it is UFO range

	END_REGION

	REGION 8 – Search window and displacement validation

	    (*Both parameters have to be checked to prevent tracking array exceeding.*)

	    // Search window cannot be lower than zero and greater than distance between PEC position and conveyor edge.
	    #sx_InvalidSearchWindow := #iUDT_PECUpdateConfiguration.SearchWindowFwd < 0
	    OR #iUDT_PECUpdateConfiguration.SearchWindowFwd >= #iUDT_ConveyorCommonConfiguration.Length + #iUDT_ConveyorCommonConfiguration.LengthCorrection - #si_PECPosition
	    OR #iUDT_PECUpdateConfiguration.SearchWindowRvs < 0
	    OR #iUDT_PECUpdateConfiguration.SearchWindowRvs >= #si_PECPosition;

	    // Displacement cannot be greater than the photoeye position.
	    IF (ABS(#si_Displacement) > #si_PECPosition)
	    THEN
	        #sx_InvalidDisplacement := TRUE;
	    END_IF;

	END_REGION

	REGION 9 – Total number of parcels counter

	    (*Parcels are counted basing on parcel detection rising edge trigger. Counting is blocked
	      during PLC first scan, when photoeye signal becomes 0.*)

	    #s_R_TRIG_Parcel(CLK := #sx_ParcelDetected);

	    IF (#s_R_TRIG_Parcel.Q
	        AND NOT "DB_Memory".FirstScan)
	    THEN
	        // Total number of parcels.
	        #sdi_TotalNumberOfParcels += 1;

	        // Every detected parcel resets lost parcels in a row counter.
	        #si_LostParcelsInARow := 0;

	        // Number of teached parcels is incremented if teaching mode is activated.
	        IF (#sx_TeachingMode)
	        THEN
	            #si_NumberOfTeachedParcels += 1;
	        END_IF;
	    END_IF;

	END_REGION

	REGION 10 – PEC Update
	    (* Photoeye position record is updated after every tracking register shift, basing on
	       actual situation - photoeye signal and data availability. In case of displacement
	       graeter than one, the loop will be executed the proper number of times. The update loop
	       can be executed if there is no configuration errors and the displacement was given.*)

	    WHILE #si_Displacement <> 0
	        AND NOT #sx_InvalidGINRange
	        AND NOT #sx_InvalidDisplacement
	        AND NOT #sx_InvalidSearchWindow
	    DO

	        REGION 10.1 – Direction

	            (*Depending on displacement sign, the direction of movement is determinated. This allows to choose
	            ` correct search window and parametrize all search loops to count up or down.*)

	            IF (#si_Displacement < 0)
	            THEN
	                #si_Direction := -1;
	                #si_SearchWindow := #iUDT_PECUpdateConfiguration.SearchWindowRvs;
	            ELSIF (#si_Displacement > 0)
	            THEN
	                #si_Direction := 1;
	                #si_SearchWindow := #iUDT_PECUpdateConfiguration.SearchWindowFwd;
	            END_IF;

	        END_REGION

	        REGION 10.2 – Position to update

	            // Position pointer used to specify the tracking array record to be updated.
	            #si_PositionToUpdate := #si_PECPosition - #si_Displacement + #si_Direction;

	        END_REGION


	        REGION 10.3 – Total number of data counter

	            (*Total number of data is incremented every time when new GIN is detected.*)

	            IF (#iqa_TrackingData[#si_PositionToUpdate + 1] > 0
	                AND #iqa_TrackingData[#si_PositionToUpdate + 1] <> #si_LastCountedData)
	            THEN
	                #sdi_TotalNumberOfData += 1;
	                #si_LastCountedData := #iqa_TrackingData[#si_PositionToUpdate + 1];
	            END_IF;

	        END_REGION

	        REGION 10.4 – GIN detection

	            (* Data found and parcel found triggers are used to determine the update case,
	               whether the data occurred first or a parcel.*)

	            // Trigger on any data found at a PEC position to detect the front of the parcel data.
	            #s_R_TRIG_DataFound(CLK := #iqa_TrackingData[#si_PositionToUpdate] <> 0);

	            // Trigger on positive data found at a PEC position to detect the front of the parcel data.
	            #s_R_TRIG_PositiveDataFound(CLK := #iqa_TrackingData[#si_PositionToUpdate] > 0);

	            // Trigger to detect front of the parcel.
	            #s_R_TRIG_ParcelFound(CLK := #sx_ParcelDetected);

	(*
	Data detected without PEC signal

